Yaskawa INFORM job: A_ROOF_SIDE_0617_2_PAINT_16.JBI

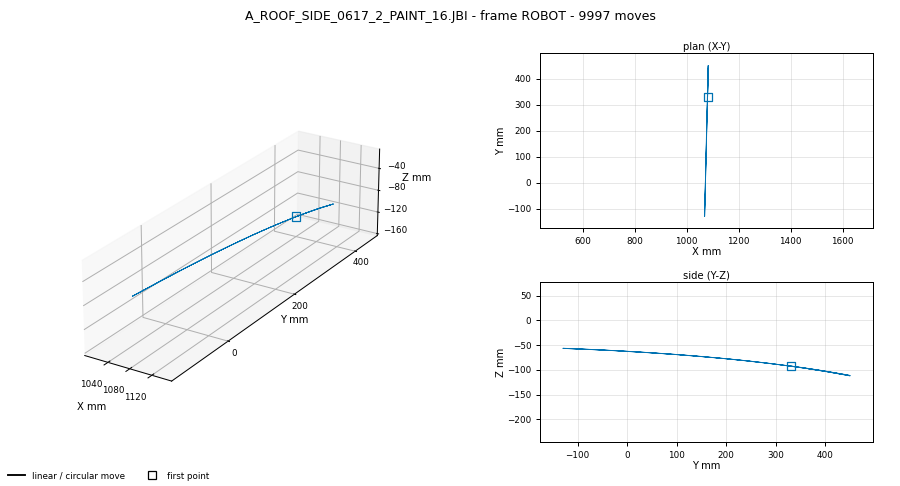
[picture p0: tool path of A_ROOF_SIDE_0617_2_PAINT_16.JBI in frame ROBOT, 9997 of 9997 moves have a stored position in this frame; points joined in program order, loops and branches not executed]
/JOB
//NAME A_ROOF_SIDE_0617_2_PAINT16
//POS
///NPOS 9997,0,0,0,0,0
///TOOL 1
///USER 0
///POSTYPE ROBOT
///RECTAN
///RCONF 1,0,0,0,0,0,0,0,0,0,0,0,0,0,0,0,0,0,0,0,0,0,0,0
C00000=1080.801,330.181,-92.181,175.912,27.090,154.615
C00001=1080.812,330.595,-92.237,175.918,27.097,154.616
C00002=1080.821,331.010,-92.293,175.923,27.105,154.617
C00003=1080.832,331.424,-92.349,175.928,27.113,154.618
C00004=1080.838,331.672,-92.382,175.931,27.117,154.619
C00005=1080.844,331.919,-92.416,175.934,27.122,154.620
C00006=1080.849,332.167,-92.449,175.937,27.126,154.620
C00007=1080.856,332.416,-92.482,175.940,27.131,154.621
C00008=1080.862,332.663,-92.516,175.943,27.136,154.622
C00009=1080.868,332.911,-92.550,175.947,27.141,154.623
C00010=1080.873,333.158,-92.584,175.950,27.146,154.623
C00011=1080.879,333.406,-92.617,175.953,27.150,154.624
C00012=1080.885,333.653,-92.651,175.956,27.155,154.625
C00013=1080.892,333.902,-92.684,175.959,27.160,154.626
C00014=1080.898,334.149,-92.718,175.962,27.165,154.627
C00015=1080.904,334.396,-92.752,175.965,27.170,154.627
C00016=1080.909,334.644,-92.786,175.968,27.174,154.628
C00017=1080.915,334.891,-92.820,175.971,27.179,154.629
C00018=1080.921,335.140,-92.853,175.975,27.183,154.630
C00019=1080.927,335.387,-92.888,175.978,27.188,154.630
C00020=1080.933,335.635,-92.922,175.981,27.193,154.631
C00021=1080.939,335.883,-92.955,175.984,27.198,154.632
C00022=1080.946,336.130,-92.989,175.987,27.202,154.633
C00023=1080.951,336.377,-93.023,175.990,27.207,154.633
C00024=1080.957,336.625,-93.056,175.994,27.212,154.634
C00025=1080.963,336.873,-93.091,175.997,27.217,154.635
C00026=1080.969,337.121,-93.125,176.000,27.222,154.636
C00027=1080.975,337.368,-93.159,176.003,27.227,154.637
C00028=1080.981,337.616,-93.192,176.006,27.232,154.637
C00029=1080.987,337.864,-93.226,176.009,27.236,154.638
C00030=1080.993,338.111,-93.260,176.012,27.241,154.639
C00031=1080.999,338.359,-93.295,176.015,27.246,154.640
C00032=1081.005,338.606,-93.329,176.018,27.251,154.641
C00033=1081.011,338.854,-93.363,176.022,27.256,154.642
C00034=1081.018,339.102,-93.397,176.025,27.261,154.642
C00035=1081.024,339.349,-93.431,176.028,27.266,154.643
C00036=1081.029,339.596,-93.466,176.031,27.270,154.644
C00037=1081.035,339.845,-93.500,176.034,27.276,154.645
C00038=1081.041,340.092,-93.534,176.037,27.280,154.646
C00039=1081.047,340.340,-93.568,176.040,27.285,154.646
C00040=1081.053,340.588,-93.602,176.043,27.290,154.647
C00041=1081.059,340.835,-93.636,176.047,27.295,154.648
C00042=1081.065,341.082,-93.671,176.050,27.300,154.649
C00043=1081.071,341.330,-93.706,176.053,27.305,154.650
C00044=1081.077,341.577,-93.740,176.056,27.310,154.650
C00045=1081.083,341.825,-93.775,176.059,27.315,154.651
C00046=1081.089,342.072,-93.809,176.062,27.320,154.652
C00047=1081.095,342.320,-93.843,176.065,27.325,154.653
C00048=1081.101,342.568,-93.877,176.069,27.330,154.654
C00049=1081.106,342.815,-93.912,176.072,27.335,154.655
C00050=1081.113,343.063,-93.946,176.075,27.340,154.655
C00051=1081.119,343.310,-93.981,176.078,27.345,154.656
C00052=1081.129,343.719,-94.038,176.084,27.353,154.658
C00053=1081.140,344.129,-94.095,176.089,27.362,154.659
C00054=1081.149,344.538,-94.152,176.095,27.370,154.660
C00055=1081.159,344.947,-94.210,176.100,27.379,154.662
C00056=1081.165,345.194,-94.244,176.103,27.383,154.663
C00057=1081.171,345.442,-94.280,176.106,27.389,154.664
C00058=1081.177,345.689,-94.314,176.109,27.394,154.665
C00059=1081.183,345.937,-94.349,176.113,27.399,154.665
C00060=1081.189,346.184,-94.383,176.116,27.404,154.666
C00061=1081.195,346.432,-94.418,176.119,27.409,154.667
C00062=1081.201,346.679,-94.453,176.122,27.414,154.668
C00063=1081.207,346.927,-94.488,176.125,27.419,154.669
C00064=1081.213,347.174,-94.523,176.129,27.425,154.670
C00065=1081.219,347.422,-94.557,176.132,27.430,154.671
C00066=1081.225,347.669,-94.593,176.135,27.435,154.671
C00067=1081.231,347.917,-94.627,176.138,27.440,154.672
C00068=1081.237,348.164,-94.663,176.142,27.446,154.673
C00069=1081.243,348.412,-94.697,176.145,27.451,154.674
C00070=1081.250,348.659,-94.732,176.148,27.456,154.675
C00071=1081.255,348.906,-94.767,176.151,27.461,154.676
C00072=1081.261,349.154,-94.802,176.154,27.466,154.677
C00073=1081.267,349.401,-94.837,176.158,27.472,154.678
C00074=1081.273,349.649,-94.873,176.161,27.477,154.679
C00075=1081.280,349.897,-94.907,176.164,27.482,154.680
C00076=1081.285,350.144,-94.943,176.167,27.488,154.680
C00077=1081.292,350.391,-94.978,176.171,27.493,154.681
C00078=1081.298,350.639,-95.013,176.174,27.498,154.682
C00079=1081.304,350.886,-95.048,176.177,27.504,154.683
C00080=1081.310,351.134,-95.083,176.181,27.509,154.684
C00081=1081.317,351.381,-95.118,176.184,27.514,154.685
C00082=1081.322,351.628,-95.154,176.187,27.519,154.686
C00083=1081.328,351.876,-95.189,176.190,27.525,154.687
C00084=1081.334,352.124,-95.224,176.194,27.530,154.688
C00085=1081.340,352.371,-95.259,176.197,27.535,154.689
C00086=1081.347,352.618,-95.294,176.200,27.541,154.689
C00087=1081.353,352.866,-95.330,176.203,27.546,154.690
C00088=1081.359,353.113,-95.366,176.207,27.552,154.691
C00089=1081.364,353.360,-95.401,176.210,27.557,154.692
C00090=1081.371,353.608,-95.436,176.213,27.562,154.693
C00091=1081.377,353.855,-95.472,176.217,27.568,154.694
C00092=1081.382,354.102,-95.508,176.220,27.573,154.695
C00093=1081.388,354.350,-95.543,176.223,27.579,154.696
C00094=1081.395,354.597,-95.578,176.227,27.584,154.697
C00095=1081.401,354.845,-95.614,176.229,27.590,154.698
C00096=1081.407,355.092,-95.650,176.232,27.595,154.699
C00097=1081.413,355.340,-95.685,176.236,27.601,154.700
C00098=1081.419,355.587,-95.721,176.239,27.606,154.701
C00099=1081.425,355.835,-95.756,176.242,27.612,154.702
C00100=1081.431,356.081,-95.792,176.246,27.617,154.703
C00101=1081.437,356.329,-95.828,176.249,27.622,154.704
C00102=1081.443,356.576,-95.864,176.252,27.628,154.705
C00103=1081.449,356.824,-95.899,176.256,27.634,154.706
C00104=1081.459,357.236,-95.959,176.261,27.643,154.707
C00105=1081.470,357.647,-96.019,176.267,27.652,154.709
C00106=1081.480,358.060,-96.078,176.272,27.661,154.711
C00107=1081.490,358.472,-96.138,176.278,27.671,154.712
C00108=1081.496,358.720,-96.174,176.281,27.676,154.713
C00109=1081.503,358.967,-96.210,176.284,27.682,154.714
C00110=1081.509,359.214,-96.245,176.288,27.688,154.715
C00111=1081.515,359.461,-96.281,176.291,27.693,154.716
C00112=1081.521,359.708,-96.317,176.294,27.699,154.717
C00113=1081.527,359.955,-96.353,176.298,27.705,154.718
C00114=1081.533,360.203,-96.389,176.301,27.711,154.719
C00115=1081.540,360.450,-96.426,176.305,27.717,154.720
C00116=1081.546,360.698,-96.461,176.308,27.722,154.721
C00117=1081.552,360.945,-96.498,176.311,27.727,154.722
C00118=1081.558,361.193,-96.533,176.315,27.733,154.723
C00119=1081.564,361.440,-96.570,176.318,27.739,154.724
C00120=1081.570,361.688,-96.606,176.322,27.745,154.725
C00121=1081.576,361.935,-96.643,176.324,27.751,154.726
C00122=1081.582,362.181,-96.679,176.327,27.756,154.727
C00123=1081.588,362.429,-96.714,176.331,27.762,154.728
C00124=1081.594,362.676,-96.751,176.334,27.768,154.729
C00125=1081.601,362.923,-96.787,176.338,27.774,154.730
C00126=1081.607,363.170,-96.823,176.341,27.780,154.731
C00127=1081.613,363.417,-96.860,176.344,27.785,154.733
C00128=1081.619,363.665,-96.896,176.348,27.792,154.734
C00129=1081.626,363.912,-96.932,176.351,27.797,154.735
C00130=1081.631,364.160,-96.969,176.355,27.803,154.736
C00131=1081.637,364.407,-97.005,176.358,27.809,154.737
C00132=1081.644,364.654,-97.042,176.362,27.815,154.738
C00133=1081.650,364.901,-97.078,176.365,27.821,154.739
C00134=1081.657,365.148,-97.115,176.369,27.827,154.740
C00135=1081.663,365.396,-97.151,176.372,27.833,154.741
C00136=1081.669,365.643,-97.188,176.374,27.839,154.742
C00137=1081.675,365.891,-97.224,176.378,27.845,154.743
C00138=1081.681,366.138,-97.261,176.381,27.850,154.744
C00139=1081.687,366.385,-97.298,176.385,27.857,154.745
C00140=1081.693,366.632,-97.334,176.388,27.862,154.746
C00141=1081.699,366.879,-97.371,176.392,27.869,154.748
C00142=1081.705,367.126,-97.408,176.395,27.875,154.749
C00143=1081.712,367.373,-97.445,176.399,27.881,154.750
C00144=1081.717,367.620,-97.482,176.402,27.887,154.751
C00145=1081.724,367.867,-97.518,176.406,27.893,154.752
C00146=1081.730,368.114,-97.555,176.409,27.899,154.753
C00147=1081.736,368.362,-97.592,176.412,27.906,154.754
C00148=1081.742,368.609,-97.628,176.415,27.911,154.755
C00149=1081.748,368.857,-97.666,176.419,27.918,154.756
C00150=1081.755,369.103,-97.703,176.422,27.924,154.758
C00151=1081.761,369.350,-97.739,176.426,27.930,154.759
C00152=1081.767,369.598,-97.776,176.429,27.936,154.760
C00153=1081.773,369.845,-97.813,176.433,27.942,154.761
C00154=1081.779,370.092,-97.850,176.436,27.948,154.762
C00155=1081.786,370.339,-97.887,176.440,27.955,154.763
C00156=1081.791,370.553,-97.919,176.443,27.960,154.764
C00157=1081.796,370.767,-97.950,176.446,27.966,154.765
C00158=1081.801,370.981,-97.983,176.448,27.970,154.766
C00159=1081.807,371.195,-98.015,176.451,27.976,154.767
C00160=1081.812,371.409,-98.047,176.454,27.981,154.768
C00161=1081.818,371.623,-98.080,176.457,27.987,154.769
C00162=1081.823,371.837,-98.112,176.460,27.992,154.770
C00163=1081.828,372.052,-98.144,176.463,27.998,154.771
C00164=1081.835,372.299,-98.181,176.467,28.004,154.772
C00165=1081.841,372.546,-98.218,176.470,28.010,154.773
C00166=1081.847,372.792,-98.255,176.474,28.016,154.775
C00167=1081.854,373.041,-98.293,176.477,28.023,154.776
C00168=1081.860,373.287,-98.330,176.480,28.030,154.777
C00169=1081.866,373.534,-98.367,176.483,28.036,154.778
C00170=1081.873,373.781,-98.404,176.487,28.042,154.779
C00171=1081.879,374.028,-98.442,176.491,28.048,154.781
C00172=1081.885,374.276,-98.479,176.494,28.055,154.782
C00173=1081.891,374.522,-98.516,176.498,28.061,154.783
C00174=1081.898,374.769,-98.555,176.501,28.068,154.784
C00175=1081.903,375.017,-98.592,176.505,28.074,154.785
C00176=1081.909,375.264,-98.629,176.508,28.081,154.787
C00177=1081.916,375.510,-98.667,176.511,28.087,154.788
C00178=1081.922,375.757,-98.705,176.515,28.094,154.789
C00179=1081.928,376.005,-98.742,176.518,28.100,154.790
C00180=1081.934,376.252,-98.779,176.522,28.107,154.792
C00181=1081.941,376.499,-98.817,176.526,28.114,154.793
C00182=1081.947,376.745,-98.855,176.529,28.120,154.794
C00183=1081.953,376.992,-98.892,176.533,28.127,154.795
C00184=1081.960,377.240,-98.931,176.535,28.133,154.797
C00185=1081.965,377.487,-98.968,176.539,28.140,154.798
C00186=1081.972,377.733,-99.005,176.543,28.146,154.799
C00187=1081.978,377.981,-99.043,176.546,28.153,154.800
C00188=1081.984,378.228,-99.081,176.550,28.160,154.802
C00189=1081.991,378.475,-99.119,176.554,28.167,154.803
C00190=1081.997,378.722,-99.157,176.557,28.173,154.804
C00191=1082.004,378.969,-99.194,176.560,28.180,154.805
C00192=1082.010,379.216,-99.232,176.564,28.187,154.807
C00193=1082.016,379.462,-99.270,176.567,28.193,154.808
C00194=1082.022,379.709,-99.308,176.571,28.200,154.809
C00195=1082.028,379.956,-99.346,176.575,28.207,154.810
C00196=1082.035,380.203,-99.384,176.578,28.214,154.812
C00197=1082.041,380.450,-99.422,176.582,28.220,154.813
C00198=1082.048,380.697,-99.460,176.585,28.227,154.814
C00199=1082.054,380.944,-99.497,176.588,28.234,154.816
C00200=1082.061,381.191,-99.536,176.592,28.241,154.817
C00201=1082.067,381.438,-99.574,176.596,28.248,154.818
C00202=1082.073,381.685,-99.612,176.599,28.255,154.820
C00203=1082.080,381.932,-99.650,176.603,28.261,154.821
C00204=1082.086,382.179,-99.689,176.606,28.268,154.822
C00205=1082.092,382.426,-99.727,176.610,28.275,154.823
C00206=1082.098,382.673,-99.765,176.613,28.282,154.825
C00207=1082.105,382.920,-99.803,176.617,28.289,154.826
C00208=1082.111,383.166,-99.841,176.621,28.296,154.827
C00209=1082.118,383.413,-99.880,176.624,28.303,154.829
C00210=1082.123,383.660,-99.918,176.627,28.310,154.830
C00211=1082.130,383.907,-99.957,176.631,28.318,154.832
C00212=1082.136,384.135,-99.993,176.634,28.324,154.833
C00213=1082.141,384.364,-100.028,176.638,28.330,154.834
C00214=1082.148,384.592,-100.063,176.641,28.337,154.835
C00215=1082.153,384.819,-100.099,176.644,28.344,154.837
C00216=1082.159,385.048,-100.135,176.648,28.350,154.838
C00217=1082.165,385.276,-100.170,176.651,28.356,154.839
C00218=1082.171,385.505,-100.206,176.655,28.363,154.840
C00219=1082.177,385.733,-100.241,176.658,28.370,154.842
C00220=1082.182,385.980,-100.280,176.661,28.377,154.843
C00221=1082.189,386.227,-100.319,176.665,28.385,154.844
C00222=1082.195,386.474,-100.357,176.668,28.392,154.846
C00223=1082.201,386.721,-100.395,176.672,28.399,154.847
C00224=1082.208,386.967,-100.434,176.676,28.406,154.849
C00225=1082.214,387.214,-100.473,176.680,28.413,154.850
C00226=1082.220,387.461,-100.512,176.683,28.421,154.852
C00227=1082.227,387.708,-100.550,176.686,28.428,154.853
C00228=1082.234,387.955,-100.589,176.690,28.435,154.854
C00229=1082.240,388.202,-100.628,176.694,28.442,154.856
C00230=1082.246,388.448,-100.667,176.698,28.450,154.857
C00231=1082.253,388.695,-100.706,176.701,28.458,154.859
C00232=1082.260,388.942,-100.744,176.705,28.465,154.860
C00233=1082.266,389.189,-100.784,176.708,28.472,154.862
C00234=1082.272,389.435,-100.822,176.712,28.479,154.863
C00235=1082.279,389.682,-100.861,176.716,28.487,154.865
C00236=1082.285,389.929,-100.901,176.719,28.494,154.866
C00237=1082.292,390.176,-100.939,176.723,28.502,154.867
C00238=1082.298,390.423,-100.978,176.727,28.509,154.869
C00239=1082.304,390.669,-101.017,176.731,28.517,154.870
C00240=1082.311,390.916,-101.056,176.734,28.524,154.872
C00241=1082.318,391.163,-101.095,176.738,28.531,154.873
C00242=1082.324,391.410,-101.134,176.741,28.539,154.875
C00243=1082.330,391.657,-101.173,176.745,28.546,154.876
C00244=1082.338,391.903,-101.213,176.749,28.554,154.878
C00245=1082.344,392.150,-101.252,176.753,28.562,154.879
C00246=1082.350,392.396,-101.291,176.756,28.570,154.881
C00247=1082.356,392.643,-101.330,176.760,28.578,154.882
C00248=1082.362,392.890,-101.370,176.763,28.585,154.884
C00249=1082.369,393.137,-101.409,176.767,28.593,154.885
C00250=1082.375,393.384,-101.449,176.771,28.601,154.887
C00251=1082.382,393.630,-101.488,176.774,28.608,154.888
C00252=1082.388,393.877,-101.528,176.778,28.616,154.890
C00253=1082.395,394.124,-101.566,176.782,28.624,154.892
C00254=1082.402,394.370,-101.607,176.786,28.632,154.893
C00255=1082.408,394.618,-101.646,176.790,28.639,154.895
C00256=1082.415,394.864,-101.686,176.793,28.647,154.896
C00257=1082.421,395.111,-101.725,176.797,28.655,154.898
C00258=1082.427,395.357,-101.765,176.801,28.663,154.899
C00259=1082.434,395.604,-101.804,176.805,28.671,154.901
C00260=1082.440,395.851,-101.844,176.808,28.679,154.903
C00261=1082.446,396.098,-101.884,176.812,28.687,154.904
C00262=1082.453,396.344,-101.924,176.816,28.695,154.906
C00263=1082.460,396.591,-101.963,176.819,28.703,154.907
C00264=1082.466,396.838,-102.003,176.823,28.711,154.909
C00265=1082.472,397.084,-102.043,176.826,28.719,154.911
C00266=1082.479,397.331,-102.082,176.830,28.727,154.912
C00267=1082.486,397.578,-102.122,176.834,28.735,154.914
C00268=1082.491,397.813,-102.161,176.838,28.743,154.915
C00269=1082.498,398.048,-102.198,176.842,28.750,154.917
C00270=1082.504,398.283,-102.236,176.845,28.759,154.919
C00271=1082.510,398.519,-102.275,176.848,28.766,154.920
C00272=1082.517,398.754,-102.313,176.852,28.774,154.922
C00273=1082.523,398.989,-102.350,176.856,28.782,154.923
C00274=1082.529,399.224,-102.389,176.860,28.790,154.925
C00275=1082.536,399.461,-102.427,176.863,28.798,154.926
C00276=1082.542,399.707,-102.467,176.867,28.806,154.928
C00277=1082.548,399.954,-102.507,176.871,28.814,154.930
C00278=1082.555,400.200,-102.547,176.875,28.823,154.932
C00279=1082.561,400.447,-102.587,176.878,28.831,154.933
C00280=1082.568,400.693,-102.628,176.882,28.840,154.935
C00281=1082.575,400.940,-102.668,176.886,28.848,154.937
C00282=1082.581,401.187,-102.708,176.890,28.856,154.938
C00283=1082.587,401.433,-102.748,176.893,28.865,154.940
C00284=1082.594,401.680,-102.789,176.897,28.873,154.942
C00285=1082.601,401.927,-102.829,176.901,28.882,154.944
C00286=1082.607,402.174,-102.869,176.905,28.890,154.945
C00287=1082.614,402.420,-102.910,176.908,28.898,154.947
C00288=1082.621,402.667,-102.951,176.913,28.907,154.949
C00289=1082.627,402.913,-102.991,176.917,28.916,154.950
C00290=1082.633,403.160,-103.031,176.921,28.924,154.952
C00291=1082.641,403.406,-103.072,176.924,28.933,154.954
C00292=1082.646,403.653,-103.113,176.928,28.942,154.956
C00293=1082.653,403.900,-103.153,176.932,28.950,154.958
C00294=1082.660,404.147,-103.193,176.936,28.959,154.959
C00295=1082.666,404.393,-103.234,176.939,28.968,154.961
C00296=1082.673,404.639,-103.274,176.944,28.976,154.963
C00297=1082.680,404.886,-103.316,176.948,28.985,154.965
C00298=1082.686,405.133,-103.356,176.952,28.994,154.967
C00299=1082.692,405.379,-103.397,176.955,29.002,154.968
C00300=1082.699,405.626,-103.438,176.959,29.012,154.970
C00301=1082.706,405.872,-103.478,176.964,29.021,154.972
C00302=1082.712,406.119,-103.520,176.968,29.030,154.974
C00303=1082.719,406.365,-103.561,176.971,29.038,154.976
C00304=1082.726,406.612,-103.601,176.975,29.047,154.978
C00305=1082.733,406.858,-103.642,176.979,29.056,154.980
C00306=1082.738,407.105,-103.683,176.983,29.065,154.981
C00307=1082.746,407.352,-103.724,176.987,29.074,154.983
C00308=1082.752,407.598,-103.765,176.991,29.083,154.985
C00309=1082.759,407.845,-103.807,176.995,29.092,154.987
C00310=1082.765,408.091,-103.847,176.999,29.102,154.989
C00311=1082.772,408.338,-103.889,177.003,29.111,154.991
C00312=1082.778,408.584,-103.930,177.007,29.120,154.993
C00313=1082.785,408.831,-103.971,177.011,29.129,154.995
C00314=1082.791,409.077,-104.012,177.015,29.139,154.997
C00315=1082.798,409.324,-104.053,177.019,29.148,154.999
C00316=1082.805,409.570,-104.094,177.023,29.157,155.001
C00317=1082.811,409.817,-104.136,177.027,29.167,155.003
C00318=1082.818,410.064,-104.177,177.031,29.176,155.004
C00319=1082.824,410.310,-104.219,177.035,29.185,155.006
C00320=1082.832,410.556,-104.260,177.040,29.195,155.008
C00321=1082.838,410.803,-104.301,177.043,29.204,155.010
C00322=1082.845,411.049,-104.343,177.047,29.213,155.012
C00323=1082.851,411.296,-104.384,177.052,29.223,155.014
C00324=1082.858,411.532,-104.424,177.056,29.232,155.016
C00325=1082.864,411.768,-104.464,177.059,29.241,155.018
C00326=1082.871,412.005,-104.504,177.063,29.250,155.020
C00327=1082.877,412.241,-104.544,177.067,29.260,155.022
C00328=1082.884,412.477,-104.583,177.072,29.269,155.024
C00329=1082.891,412.713,-104.624,177.075,29.278,155.026
C00330=1082.897,412.949,-104.663,177.079,29.287,155.028
C00331=1082.903,413.186,-104.703,177.083,29.296,155.030
C00332=1082.910,413.432,-104.746,177.088,29.306,155.032
C00333=1082.917,413.678,-104.787,177.091,29.316,155.034
C00334=1082.923,413.925,-104.828,177.096,29.326,155.036
C00335=1082.931,414.171,-104.870,177.100,29.335,155.038
C00336=1082.937,414.418,-104.912,177.104,29.345,155.040
C00337=1082.944,414.664,-104.955,177.108,29.355,155.042
C00338=1082.951,414.910,-104.995,177.112,29.365,155.044
C00339=1082.958,415.156,-105.038,177.117,29.375,155.046
C00340=1082.964,415.403,-105.080,177.120,29.384,155.048
C00341=1082.972,415.649,-105.122,177.125,29.394,155.051
C00342=1082.979,415.896,-105.164,177.129,29.404,155.053
C00343=1082.985,416.142,-105.206,177.134,29.414,155.055
C00344=1082.992,416.389,-105.248,177.137,29.424,155.057
C00345=1082.998,416.635,-105.290,177.142,29.435,155.059
C00346=1083.005,416.881,-105.333,177.147,29.445,155.061
C00347=1083.013,417.127,-105.375,177.150,29.455,155.063
C00348=1083.019,417.374,-105.416,177.155,29.465,155.066
C00349=1083.026,417.620,-105.459,177.159,29.476,155.068
C00350=1083.033,417.867,-105.502,177.163,29.486,155.070
C00351=1083.040,418.113,-105.544,177.167,29.496,155.072
C00352=1083.046,418.359,-105.586,177.172,29.506,155.074
C00353=1083.053,418.605,-105.629,177.177,29.517,155.077
C00354=1083.060,418.851,-105.671,177.180,29.527,155.079
C00355=1083.066,419.098,-105.713,177.185,29.538,155.081
C00356=1083.073,419.344,-105.756,177.190,29.548,155.083
C00357=1083.080,419.591,-105.798,177.193,29.558,155.086
C00358=1083.087,419.836,-105.842,177.198,29.569,155.088
C00359=1083.094,420.083,-105.884,177.202,29.580,155.090
C00360=1083.101,420.329,-105.927,177.207,29.590,155.092
C00361=1083.108,420.575,-105.969,177.211,29.600,155.095
C00362=1083.115,420.821,-106.012,177.215,29.611,155.097
C00363=1083.121,421.068,-106.054,177.220,29.622,155.099
C00364=1083.129,421.315,-106.097,177.224,29.632,155.102
C00365=1083.136,421.560,-106.140,177.229,29.644,155.104
C00366=1083.143,421.807,-106.183,177.233,29.654,155.106
C00367=1083.150,422.053,-106.225,177.238,29.665,155.109
C00368=1083.157,422.299,-106.269,177.242,29.676,155.111
C00369=1083.164,422.545,-106.311,177.247,29.687,155.113
C00370=1083.171,422.791,-106.354,177.251,29.698,155.116
C00371=1083.177,423.037,-106.398,177.255,29.708,155.118
C00372=1083.184,423.283,-106.440,177.260,29.719,155.120
C00373=1083.191,423.529,-106.483,177.265,29.731,155.123
C00374=1083.199,423.776,-106.526,177.268,29.741,155.125
C00375=1083.205,424.022,-106.570,177.273,29.753,155.128
C00376=1083.212,424.268,-106.613,177.278,29.764,155.130
C00377=1083.219,424.514,-106.656,177.283,29.775,155.133
C00378=1083.225,424.760,-106.700,177.287,29.786,155.135
C00379=1083.233,425.007,-106.743,177.291,29.797,155.138
C00380=1083.240,425.254,-106.787,177.296,29.809,155.140
C00381=1083.247,425.501,-106.830,177.300,29.820,155.142
C00382=1083.254,425.748,-106.873,177.305,29.831,155.145
C00383=1083.261,425.995,-106.917,177.310,29.843,155.147
C00384=1083.268,426.241,-106.960,177.315,29.854,155.150
C00385=1083.275,426.487,-107.003,177.319,29.866,155.152
C00386=1083.282,426.733,-107.048,177.324,29.877,155.155
C00387=1083.289,426.979,-107.091,177.329,29.888,155.157
C00388=1083.296,427.225,-107.134,177.332,29.900,155.160
C00389=1083.304,427.471,-107.178,177.337,29.911,155.163
C00390=1083.311,427.717,-107.222,177.342,29.923,155.165
C00391=1083.317,427.963,-107.265,177.347,29.935,155.168
C00392=1083.325,428.209,-107.309,177.351,29.947,155.170
C00393=1083.332,428.455,-107.352,177.356,29.958,155.173
C00394=1083.339,428.702,-107.397,177.361,29.970,155.175
C00395=1083.345,428.948,-107.440,177.366,29.982,155.178
C00396=1083.353,429.193,-107.484,177.370,29.994,155.181
C00397=1083.360,429.439,-107.529,177.375,30.006,155.183
C00398=1083.367,429.685,-107.572,177.380,30.018,155.186
C00399=1083.374,429.932,-107.616,177.384,30.030,155.189
C00400=1083.382,430.177,-107.660,177.389,30.042,155.191
C00401=1083.388,430.423,-107.704,177.394,30.054,155.194
C00402=1083.395,430.669,-107.749,177.399,30.066,155.197
C00403=1083.403,430.914,-107.792,177.403,30.078,155.199
C00404=1083.410,431.160,-107.837,177.408,30.090,155.202
C00405=1083.417,431.406,-107.880,177.413,30.102,155.205
C00406=1083.424,431.652,-107.925,177.418,30.114,155.208
C00407=1083.431,431.899,-107.969,177.423,30.127,155.210
C00408=1083.439,432.144,-108.013,177.428,30.139,155.213
C00409=1083.446,432.391,-108.058,177.433,30.152,155.216
C00410=1083.453,432.636,-108.102,177.438,30.164,155.218
C00411=1083.460,432.882,-108.147,177.442,30.176,155.221
C00412=1083.466,433.128,-108.191,177.447,30.189,155.224
C00413=1083.474,433.374,-108.235,177.452,30.202,155.227
C00414=1083.482,433.620,-108.280,177.457,30.214,155.230
C00415=1083.489,433.865,-108.325,177.462,30.227,155.233
C00416=1083.496,434.111,-108.370,177.467,30.239,155.235
C00417=1083.503,434.356,-108.414,177.472,30.252,155.238
C00418=1083.510,434.602,-108.459,177.477,30.265,155.241
C00419=1083.517,434.849,-108.504,177.481,30.278,155.244
C00420=1083.524,435.092,-108.548,177.486,30.291,155.247
C00421=1083.531,435.335,-108.592,177.492,30.303,155.250
C00422=1083.538,435.579,-108.637,177.497,30.316,155.253
C00423=1083.545,435.823,-108.681,177.501,30.329,155.256
C00424=1083.553,436.066,-108.726,177.506,30.342,155.259
C00425=1083.560,436.309,-108.770,177.511,30.355,155.261
C00426=1083.567,436.553,-108.815,177.517,30.368,155.264
C00427=1083.575,436.796,-108.860,177.522,30.381,155.267
C00428=1083.582,437.042,-108.905,177.526,30.394,155.270
C00429=1083.589,437.288,-108.950,177.531,30.407,155.273
C00430=1083.596,437.533,-108.995,177.537,30.421,155.276
C00431=1083.604,437.779,-109.040,177.542,30.434,155.279
C00432=1083.611,438.025,-109.085,177.547,30.447,155.283
C00433=1083.619,438.270,-109.130,177.552,30.460,155.285
C00434=1083.626,438.517,-109.175,177.557,30.474,155.289
C00435=1083.634,438.762,-109.221,177.563,30.487,155.292
C00436=1083.644,439.107,-109.284,177.569,30.507,155.296
C00437=1083.655,439.451,-109.348,177.577,30.525,155.300
C00438=1083.665,439.796,-109.412,177.584,30.545,155.305
C00439=1083.676,440.141,-109.476,177.591,30.564,155.309
C00440=1083.683,440.386,-109.521,177.597,30.578,155.312
C00441=1083.690,440.631,-109.567,177.602,30.592,155.315
C00442=1083.697,440.877,-109.612,177.608,30.606,155.319
C00443=1083.704,441.123,-109.658,177.613,30.620,155.322
C00444=1083.712,441.368,-109.704,177.618,30.634,155.325
C00445=1083.720,441.614,-109.750,177.623,30.648,155.328
C00446=1083.727,441.860,-109.796,177.629,30.662,155.332
C00447=1083.735,442.106,-109.841,177.634,30.676,155.335
C00448=1083.743,442.351,-109.887,177.640,30.691,155.338
C00449=1083.749,442.597,-109.933,177.645,30.705,155.342
C00450=1083.757,442.842,-109.980,177.650,30.719,155.345
C00451=1083.764,443.087,-110.026,177.655,30.733,155.348
C00452=1083.772,443.333,-110.072,177.661,30.748,155.351
C00453=1083.780,443.578,-110.117,177.667,30.763,155.355
C00454=1083.786,443.824,-110.163,177.672,30.777,155.358
C00455=1083.795,444.069,-110.210,177.678,30.792,155.362
C00456=1083.802,444.315,-110.256,177.683,30.806,155.365
C00457=1083.810,444.560,-110.303,177.689,30.821,155.368
C00458=1083.817,444.805,-110.348,177.694,30.836,155.372
C00459=1083.825,445.052,-110.395,177.699,30.851,155.375
C00460=1083.833,445.297,-110.441,177.705,30.866,155.379
C00461=1083.840,445.542,-110.488,177.711,30.881,155.382
C00462=1083.847,445.788,-110.535,177.716,30.895,155.386
C00463=1083.856,446.033,-110.581,177.721,30.910,155.389
C00464=1083.862,446.279,-110.628,177.725,30.925,155.393
C00465=1083.870,446.524,-110.674,177.730,30.940,155.396
C00466=1083.878,446.769,-110.721,177.734,30.955,155.400
C00467=1083.885,447.015,-110.768,177.738,30.969,155.403
C00468=1083.893,447.260,-110.814,177.742,30.984,155.407
C00469=1083.901,447.506,-110.861,177.746,30.999,155.410
C00470=1083.909,447.751,-110.908,177.749,31.014,155.414
C00471=1083.917,447.996,-110.955,177.752,31.028,155.418
C00472=1083.924,448.242,-111.002,177.755,31.044,155.421
C00473=1083.932,448.486,-111.048,177.758,31.058,155.425
C00474=1083.940,448.732,-111.096,177.760,31.073,155.428
C00475=1083.947,448.977,-111.143,177.763,31.088,155.432
C00476=1083.955,449.222,-111.189,177.765,31.102,155.436
C00477=1083.963,449.468,-111.236,177.767,31.117,155.439
C00478=1083.973,449.712,-111.281,177.770,31.130,155.443
C00479=1083.985,449.959,-111.326,177.772,31.143,155.446
C00480=1083.614,449.951,-111.536,177.739,31.321,155.494
C00481=1083.601,449.705,-111.492,177.737,31.309,155.490
C00482=1083.591,449.459,-111.446,177.735,31.295,155.487
C00483=1083.583,449.215,-111.400,177.733,31.281,155.483
C00484=1083.575,448.969,-111.353,177.730,31.266,155.480
C00485=1083.567,448.725,-111.306,177.728,31.251,155.476
C00486=1083.559,448.479,-111.258,177.725,31.236,155.473
C00487=1083.552,448.234,-111.211,177.722,31.222,155.469
C00488=1083.544,447.989,-111.165,177.719,31.207,155.465
C00489=1083.536,447.744,-111.118,177.716,31.192,155.462
C00490=1083.529,447.497,-111.071,177.712,31.177,155.458
C00491=1083.521,447.252,-111.025,177.708,31.162,155.454
C00492=1083.513,447.007,-110.977,177.704,31.147,155.451
C00493=1083.506,446.761,-110.930,177.700,31.132,155.447
C00494=1083.497,446.516,-110.884,177.696,31.118,155.444
C00495=1083.490,446.271,-110.837,177.691,31.103,155.440
C00496=1083.483,446.025,-110.791,177.687,31.088,155.437
C00497=1083.475,445.780,-110.744,177.682,31.073,155.433
C00498=1083.468,445.534,-110.697,177.676,31.058,155.430
C00499=1083.460,445.289,-110.651,177.671,31.044,155.426
C00500=1083.453,445.044,-110.604,177.665,31.028,155.423
C00501=1083.444,444.798,-110.557,177.660,31.014,155.419
C00502=1083.437,444.553,-110.511,177.654,30.999,155.416
C00503=1083.429,444.308,-110.465,177.648,30.984,155.412
C00504=1083.421,444.062,-110.419,177.643,30.969,155.409
C00505=1083.414,443.816,-110.373,177.637,30.955,155.406
C00506=1083.406,443.571,-110.326,177.631,30.940,155.402
C00507=1083.399,443.325,-110.280,177.626,30.926,155.399
C00508=1083.392,443.080,-110.234,177.620,30.911,155.396
C00509=1083.384,442.834,-110.187,177.615,30.897,155.392
C00510=1083.376,442.589,-110.141,177.609,30.883,155.389
C00511=1083.369,442.343,-110.096,177.604,30.868,155.386
C00512=1083.362,442.098,-110.049,177.598,30.854,155.382
C00513=1083.354,441.852,-110.004,177.593,30.840,155.379
C00514=1083.346,441.607,-109.958,177.587,30.826,155.376
C00515=1083.340,441.361,-109.912,177.582,30.811,155.372
C00516=1083.332,441.116,-109.866,177.577,30.797,155.369
C00517=1083.324,440.870,-109.821,177.572,30.784,155.366
C00518=1083.317,440.625,-109.775,177.566,30.770,155.363
C00519=1083.310,440.379,-109.729,177.561,30.756,155.360
C00520=1083.302,440.133,-109.683,177.555,30.742,155.357
C00521=1083.292,439.804,-109.622,177.548,30.723,155.352
C00522=1083.282,439.474,-109.561,177.541,30.705,155.348
C00523=1083.272,439.145,-109.500,177.534,30.687,155.344
C00524=1083.262,438.816,-109.440,177.527,30.668,155.340
C00525=1083.254,438.571,-109.394,177.522,30.655,155.337
C00526=1083.247,438.325,-109.348,177.516,30.641,155.334
C00527=1083.239,438.079,-109.303,177.511,30.628,155.331
C00528=1083.232,437.834,-109.258,177.506,30.615,155.327
C00529=1083.224,437.588,-109.213,177.500,30.601,155.324
C00530=1083.217,437.342,-109.168,177.495,30.588,155.321
C00531=1083.209,437.096,-109.122,177.491,30.575,155.318
C00532=1083.202,436.850,-109.077,177.485,30.561,155.315
C00533=1083.195,436.606,-109.032,177.480,30.548,155.312
C00534=1083.188,436.359,-108.987,177.475,30.535,155.309
C00535=1083.180,436.113,-108.942,177.470,30.522,155.306
C00536=1083.173,435.867,-108.897,177.464,30.509,155.303
C00537=1083.165,435.622,-108.852,177.459,30.496,155.301
C00538=1083.159,435.377,-108.807,177.454,30.483,155.298
C00539=1083.151,435.131,-108.762,177.450,30.470,155.295
C00540=1083.144,434.884,-108.717,177.444,30.457,155.292
C00541=1083.137,434.639,-108.673,177.439,30.445,155.289
C00542=1083.130,434.393,-108.628,177.434,30.432,155.286
C00543=1083.123,434.147,-108.583,177.429,30.419,155.283
C00544=1083.116,433.902,-108.538,177.424,30.406,155.280
C00545=1083.108,433.656,-108.494,177.420,30.394,155.277
C00546=1083.100,433.410,-108.449,177.414,30.381,155.275
C00547=1083.094,433.164,-108.404,177.409,30.368,155.272
C00548=1083.087,432.918,-108.360,177.404,30.356,155.269
C00549=1083.080,432.672,-108.315,177.399,30.343,155.266
C00550=1083.073,432.426,-108.271,177.394,30.331,155.263
C00551=1083.065,432.181,-108.226,177.390,30.318,155.261
C00552=1083.058,431.935,-108.182,177.385,30.306,155.258
C00553=1083.051,431.689,-108.137,177.380,30.294,155.255
C00554=1083.043,431.443,-108.093,177.375,30.282,155.252
C00555=1083.036,431.197,-108.049,177.370,30.269,155.250
C00556=1083.029,430.951,-108.004,177.365,30.257,155.247
C00557=1083.022,430.705,-107.961,177.360,30.245,155.244
C00558=1083.014,430.459,-107.916,177.355,30.233,155.242
C00559=1083.008,430.213,-107.872,177.350,30.221,155.239
C00560=1083.000,429.967,-107.828,177.345,30.209,155.236
C00561=1082.994,429.721,-107.784,177.340,30.197,155.233
C00562=1082.986,429.475,-107.740,177.336,30.185,155.231
C00563=1082.979,429.230,-107.696,177.331,30.173,155.228
C00564=1082.972,428.984,-107.653,177.326,30.161,155.225
C00565=1082.965,428.737,-107.608,177.321,30.149,155.223
C00566=1082.958,428.491,-107.565,177.317,30.137,155.220
C00567=1082.951,428.245,-107.521,177.313,30.126,155.218
C00568=1082.944,428.000,-107.476,177.308,30.114,155.215
C00569=1082.936,427.753,-107.433,177.303,30.102,155.212
C00570=1082.929,427.508,-107.390,177.298,30.090,155.210
C00571=1082.923,427.262,-107.346,177.293,30.079,155.207
C00572=1082.915,427.015,-107.302,177.289,30.067,155.205
C00573=1082.908,426.770,-107.259,177.284,30.056,155.202
C00574=1082.901,426.525,-107.215,177.279,30.044,155.200
C00575=1082.894,426.280,-107.172,177.274,30.033,155.197
C00576=1082.887,426.035,-107.128,177.270,30.022,155.195
C00577=1082.880,425.790,-107.085,177.266,30.010,155.192
C00578=1082.873,425.546,-107.042,177.261,29.999,155.190
C00579=1082.865,425.301,-106.999,177.256,29.988,155.187
C00580=1082.859,425.056,-106.956,177.251,29.977,155.185
C00581=1082.852,424.810,-106.912,177.246,29.965,155.182
C00582=1082.845,424.563,-106.869,177.243,29.954,155.180
C00583=1082.838,424.317,-106.826,177.238,29.943,155.177
C00584=1082.831,424.072,-106.783,177.233,29.932,155.175
C00585=1082.824,423.826,-106.739,177.228,29.921,155.173
C00586=1082.817,423.579,-106.697,177.223,29.909,155.170
C00587=1082.810,423.333,-106.653,177.220,29.899,155.168
C00588=1082.803,423.087,-106.610,177.215,29.887,155.165
C00589=1082.796,422.841,-106.567,177.210,29.876,155.163
C00590=1082.789,422.594,-106.524,177.205,29.866,155.161
C00591=1082.782,422.349,-106.481,177.202,29.855,155.158
C00592=1082.775,422.102,-106.438,177.197,29.843,155.156
C00593=1082.764,421.711,-106.369,177.190,29.827,155.152
C00594=1082.753,421.319,-106.302,177.183,29.809,155.148
C00595=1082.742,420.927,-106.234,177.176,29.793,155.145
C00596=1082.731,420.536,-106.165,177.169,29.775,155.141
C00597=1082.724,420.289,-106.123,177.164,29.765,155.139
C00598=1082.717,420.043,-106.080,177.159,29.754,155.136
C00599=1082.710,419.797,-106.038,177.155,29.744,155.134
C00600=1082.703,419.551,-105.995,177.150,29.733,155.132
C00601=1082.696,419.304,-105.953,177.147,29.723,155.130
C00602=1082.690,419.058,-105.910,177.142,29.712,155.127
C00603=1082.683,418.812,-105.868,177.137,29.702,155.125
C00604=1082.676,418.565,-105.825,177.133,29.691,155.123
C00605=1082.669,418.319,-105.782,177.129,29.681,155.121
C00606=1082.662,418.073,-105.740,177.124,29.670,155.118
C00607=1082.655,417.827,-105.697,177.120,29.660,155.116
C00608=1082.648,417.580,-105.655,177.115,29.650,155.114
C00609=1082.642,417.334,-105.612,177.111,29.640,155.112
C00610=1082.635,417.088,-105.570,177.107,29.629,155.110
C00611=1082.628,416.842,-105.529,177.103,29.619,155.108
C00612=1082.621,416.596,-105.486,177.098,29.609,155.105
C00613=1082.614,416.349,-105.444,177.094,29.599,155.103
C00614=1082.607,416.103,-105.401,177.090,29.589,155.101
C00615=1082.601,415.856,-105.359,177.086,29.579,155.099
C00616=1082.594,415.610,-105.317,177.081,29.569,155.097
C00617=1082.586,415.364,-105.275,177.077,29.559,155.095
C00618=1082.581,415.118,-105.233,177.072,29.549,155.093
C00619=1082.574,414.871,-105.191,177.069,29.539,155.090
C00620=1082.566,414.625,-105.150,177.064,29.530,155.088
C00621=1082.560,414.378,-105.107,177.060,29.519,155.086
C00622=1082.553,414.132,-105.065,177.055,29.510,155.084
C00623=1082.545,413.886,-105.023,177.052,29.500,155.082
C00624=1082.539,413.639,-104.982,177.047,29.490,155.080
C00625=1082.532,413.393,-104.941,177.043,29.481,155.078
C00626=1082.525,413.147,-104.898,177.039,29.471,155.076
C00627=1082.519,412.900,-104.856,177.034,29.461,155.074
C00628=1082.512,412.654,-104.815,177.031,29.452,155.072
C00629=1082.503,412.325,-104.759,177.025,29.439,155.069
C00630=1082.494,411.997,-104.704,177.019,29.426,155.067
C00631=1082.484,411.669,-104.648,177.014,29.413,155.064
C00632=1082.476,411.340,-104.593,177.008,29.401,155.061
C00633=1082.469,411.093,-104.551,177.004,29.391,155.059
C00634=1082.462,410.848,-104.511,177.000,29.382,155.057
C00635=1082.456,410.601,-104.469,176.996,29.372,155.055
C00636=1082.449,410.355,-104.428,176.992,29.363,155.053
C00637=1082.442,410.108,-104.385,176.987,29.353,155.051
C00638=1082.435,409.862,-104.344,176.983,29.344,155.049
C00639=1082.429,409.616,-104.303,176.980,29.335,155.047
C00640=1082.422,409.368,-104.262,176.975,29.325,155.045
C00641=1082.416,409.122,-104.221,176.971,29.316,155.043
C00642=1082.409,408.876,-104.180,176.967,29.307,155.041
C00643=1082.403,408.629,-104.138,176.964,29.298,155.040
C00644=1082.396,408.383,-104.097,176.959,29.288,155.038
C00645=1082.389,408.137,-104.056,176.955,29.279,155.036
C00646=1082.382,407.890,-104.014,176.951,29.270,155.034
C00647=1082.376,407.644,-103.974,176.947,29.261,155.032
C00648=1082.370,407.397,-103.932,176.943,29.252,155.030
C00649=1082.363,407.151,-103.891,176.939,29.243,155.028
C00650=1082.356,406.904,-103.850,176.935,29.234,155.026
C00651=1082.350,406.657,-103.809,176.931,29.225,155.024
C00652=1082.343,406.411,-103.768,176.928,29.216,155.022
C00653=1082.336,406.164,-103.728,176.923,29.206,155.020
C00654=1082.330,405.917,-103.686,176.919,29.198,155.019
C00655=1082.323,405.671,-103.645,176.915,29.189,155.017
C00656=1082.316,405.424,-103.605,176.911,29.180,155.015
C00657=1082.309,405.178,-103.564,176.908,29.171,155.013
C00658=1082.303,404.931,-103.523,176.903,29.162,155.011
C00659=1082.296,404.685,-103.482,176.899,29.153,155.010
C00660=1082.290,404.438,-103.442,176.895,29.145,155.008
C00661=1082.283,404.191,-103.401,176.891,29.136,155.006
C00662=1082.276,403.945,-103.360,176.888,29.127,155.004
C00663=1082.270,403.698,-103.319,176.884,29.119,155.002
C00664=1082.264,403.451,-103.279,176.880,29.110,155.001
C00665=1082.257,403.205,-103.238,176.875,29.101,154.999
C00666=1082.250,402.958,-103.198,176.871,29.092,154.997
C00667=1082.244,402.712,-103.158,176.868,29.084,154.995
C00668=1082.237,402.466,-103.117,176.864,29.076,154.994
C00669=1082.230,402.218,-103.076,176.860,29.067,154.992
C00670=1082.224,401.972,-103.036,176.856,29.058,154.990
C00671=1082.217,401.725,-102.996,176.852,29.050,154.988
C00672=1082.211,401.479,-102.956,176.849,29.041,154.986
C00673=1082.204,401.232,-102.915,176.845,29.033,154.985
C00674=1082.198,400.985,-102.875,176.841,29.025,154.983
C00675=1082.191,400.739,-102.834,176.837,29.016,154.981
C00676=1082.184,400.493,-102.794,176.833,29.008,154.980
C00677=1082.177,400.246,-102.754,176.830,28.999,154.978
C00678=1082.171,399.999,-102.713,176.826,28.991,154.976
C00679=1082.165,399.753,-102.673,176.822,28.983,154.974
C00680=1082.158,399.506,-102.633,176.817,28.974,154.973
C00681=1082.152,399.270,-102.595,176.814,28.966,154.971
C00682=1082.145,399.034,-102.557,176.810,28.958,154.970
C00683=1082.140,398.798,-102.519,176.807,28.951,154.968
C00684=1082.134,398.562,-102.480,176.803,28.943,154.966
C00685=1082.127,398.326,-102.442,176.800,28.935,154.965
C00686=1082.121,398.090,-102.404,176.796,28.927,154.963
C00687=1082.114,397.854,-102.366,176.792,28.919,154.962
C00688=1082.108,397.618,-102.327,176.788,28.911,154.960
C00689=1082.102,397.371,-102.288,176.784,28.903,154.958
C00690=1082.095,397.125,-102.248,176.781,28.895,154.957
C00691=1082.088,396.878,-102.208,176.777,28.887,154.955
C00692=1082.082,396.631,-102.168,176.773,28.879,154.954
C00693=1082.076,396.385,-102.128,176.769,28.871,154.952
C00694=1082.069,396.139,-102.089,176.766,28.863,154.950
C00695=1082.063,395.891,-102.049,176.762,28.855,154.949
C00696=1082.056,395.645,-102.009,176.759,28.847,154.947
C00697=1082.050,395.398,-101.970,176.755,28.839,154.945
C00698=1082.043,395.152,-101.930,176.751,28.831,154.944
C00699=1082.037,394.905,-101.890,176.747,28.823,154.942
C00700=1082.031,394.658,-101.851,176.743,28.816,154.941
C00701=1082.024,394.411,-101.812,176.739,28.808,154.939
C00702=1082.018,394.165,-101.772,176.736,28.800,154.938
C00703=1082.012,393.918,-101.732,176.732,28.792,154.936
C00704=1082.004,393.671,-101.693,176.728,28.784,154.934
C00705=1081.998,393.424,-101.653,176.724,28.776,154.933
C00706=1081.991,393.178,-101.614,176.721,28.769,154.931
C00707=1081.985,392.931,-101.574,176.717,28.761,154.930
C00708=1081.978,392.684,-101.535,176.714,28.753,154.928
C00709=1081.972,392.437,-101.496,176.710,28.746,154.927
C00710=1081.965,392.191,-101.456,176.706,28.738,154.925
C00711=1081.959,391.944,-101.417,176.702,28.730,154.924
C00712=1081.954,391.697,-101.378,176.698,28.723,154.922
C00713=1081.947,391.450,-101.339,176.694,28.715,154.921
C00714=1081.940,391.204,-101.299,176.692,28.707,154.919
C00715=1081.934,390.957,-101.260,176.688,28.700,154.918
C00716=1081.927,390.710,-101.221,176.684,28.692,154.916
C00717=1081.920,390.463,-101.182,176.680,28.685,154.915
C00718=1081.914,390.216,-101.143,176.676,28.677,154.913
C00719=1081.907,389.969,-101.104,176.672,28.670,154.912
C00720=1081.901,389.723,-101.066,176.669,28.662,154.910
C00721=1081.895,389.476,-101.026,176.666,28.655,154.909
C00722=1081.888,389.229,-100.987,176.662,28.648,154.907
C00723=1081.881,388.982,-100.949,176.658,28.640,154.906
C00724=1081.874,388.736,-100.910,176.654,28.633,154.905
C00725=1081.869,388.489,-100.871,176.650,28.625,154.903
C00726=1081.862,388.242,-100.832,176.646,28.618,154.902
C00727=1081.855,387.996,-100.793,176.644,28.611,154.900
C00728=1081.849,387.748,-100.754,176.640,28.604,154.899
C00729=1081.843,387.502,-100.715,176.636,28.596,154.897
C00730=1081.836,387.255,-100.677,176.632,28.589,154.896
C00731=1081.830,387.008,-100.638,176.628,28.581,154.895
C00732=1081.823,386.762,-100.600,176.625,28.574,154.893
C00733=1081.817,386.515,-100.560,176.621,28.567,154.892
C00734=1081.811,386.268,-100.521,176.618,28.560,154.890
C00735=1081.805,386.021,-100.484,176.614,28.552,154.889
C00736=1081.798,385.774,-100.445,176.611,28.546,154.888
C00737=1081.792,385.545,-100.408,176.607,28.539,154.886
C00738=1081.786,385.317,-100.373,176.604,28.532,154.885
C00739=1081.780,385.087,-100.337,176.600,28.526,154.884
C00740=1081.775,384.859,-100.302,176.597,28.519,154.882
C00741=1081.768,384.630,-100.266,176.594,28.513,154.881
C00742=1081.762,384.402,-100.230,176.590,28.506,154.880
C00743=1081.757,384.172,-100.194,176.587,28.499,154.879
C00744=1081.751,383.943,-100.159,176.583,28.492,154.877
C00745=1081.745,383.696,-100.120,176.580,28.485,154.876
C00746=1081.739,383.450,-100.082,176.576,28.478,154.875
C00747=1081.732,383.203,-100.043,176.573,28.471,154.873
C00748=1081.726,382.956,-100.005,176.570,28.465,154.872
C00749=1081.720,382.708,-99.967,176.566,28.457,154.870
C00750=1081.714,382.462,-99.928,176.562,28.450,154.869
C00751=1081.707,382.215,-99.890,176.558,28.443,154.868
C00752=1081.701,381.969,-99.852,176.555,28.437,154.866
C00753=1081.695,381.721,-99.814,176.551,28.429,154.865
C00754=1081.689,381.475,-99.776,176.547,28.422,154.864
C00755=1081.682,381.227,-99.738,176.545,28.416,154.862
C00756=1081.675,380.981,-99.700,176.541,28.409,154.861
C00757=1081.669,380.734,-99.662,176.537,28.402,154.860
C00758=1081.662,380.486,-99.624,176.534,28.396,154.859
C00759=1081.656,380.240,-99.586,176.530,28.388,154.857
C00760=1081.650,379.993,-99.547,176.526,28.381,154.856
C00761=1081.644,379.746,-99.509,176.523,28.375,154.855
C00762=1081.637,379.499,-99.471,176.519,28.368,154.853
C00763=1081.631,379.252,-99.434,176.515,28.361,154.852
C00764=1081.625,379.005,-99.396,176.513,28.355,154.851
C00765=1081.618,378.758,-99.358,176.509,28.348,154.850
C00766=1081.612,378.511,-99.320,176.505,28.341,154.848
C00767=1081.606,378.264,-99.282,176.502,28.335,154.847
C00768=1081.600,378.017,-99.244,176.498,28.328,154.846
C00769=1081.593,377.770,-99.207,176.495,28.321,154.845
C00770=1081.587,377.523,-99.169,176.491,28.315,154.843
C00771=1081.581,377.276,-99.131,176.487,28.308,154.842
C00772=1081.574,377.029,-99.093,176.484,28.302,154.841
C00773=1081.568,376.782,-99.056,176.480,28.295,154.840
C00774=1081.561,376.535,-99.018,176.478,28.288,154.838
C00775=1081.555,376.288,-98.980,176.474,28.282,154.837
C00776=1081.550,376.041,-98.943,176.470,28.275,154.836
C00777=1081.543,375.794,-98.905,176.467,28.268,154.834
C00778=1081.537,375.547,-98.867,176.463,28.262,154.833
C00779=1081.531,375.300,-98.830,176.460,28.255,154.832
C00780=1081.525,375.054,-98.792,176.456,28.249,154.831
C00781=1081.519,374.806,-98.755,176.452,28.242,154.830
C00782=1081.513,374.559,-98.717,176.449,28.236,154.828
C00783=1081.506,374.312,-98.680,176.445,28.229,154.827
C00784=1081.500,374.064,-98.643,176.442,28.223,154.826
C00785=1081.494,373.818,-98.605,176.439,28.216,154.825
C00786=1081.487,373.571,-98.568,176.436,28.210,154.824
C00787=1081.481,373.323,-98.530,176.432,28.204,154.822
C00788=1081.474,373.077,-98.493,176.429,28.198,154.821
C00789=1081.469,372.829,-98.456,176.425,28.191,154.820
C00790=1081.462,372.582,-98.419,176.421,28.184,154.819
C00791=1081.456,372.335,-98.382,176.418,28.178,154.818
C00792=1081.449,372.088,-98.344,176.414,28.172,154.817
C00793=1081.444,371.874,-98.312,176.411,28.166,154.815
C00794=1081.438,371.659,-98.280,176.408,28.161,154.815
C00795=1081.433,371.444,-98.248,176.406,28.156,154.813
C00796=1081.427,371.229,-98.215,176.403,28.150,154.812
C00797=1081.423,371.015,-98.183,176.400,28.145,154.812
C00798=1081.417,370.800,-98.151,176.397,28.139,154.810
C00799=1081.412,370.585,-98.119,176.394,28.134,154.809
C00800=1081.406,370.371,-98.086,176.390,28.129,154.809
C00801=1081.400,370.124,-98.049,176.387,28.122,154.807
C00802=1081.394,369.877,-98.012,176.384,28.116,154.806
C00803=1081.388,369.630,-97.976,176.380,28.110,154.805
C00804=1081.381,369.383,-97.939,176.377,28.104,154.804
C00805=1081.375,369.135,-97.901,176.373,28.097,154.803
C00806=1081.368,368.888,-97.865,176.370,28.092,154.802
C00807=1081.363,368.641,-97.828,176.366,28.085,154.801
C00808=1081.357,368.394,-97.791,176.363,28.079,154.799
C00809=1081.350,368.147,-97.754,176.360,28.073,154.798
C00810=1081.344,367.900,-97.717,176.356,28.067,154.797
C00811=1081.338,367.653,-97.681,176.353,28.061,154.796
C00812=1081.332,367.406,-97.644,176.349,28.054,154.795
C00813=1081.325,367.158,-97.607,176.346,28.049,154.794
C00814=1081.319,366.911,-97.570,176.342,28.042,154.793
C00815=1081.314,366.663,-97.533,176.339,28.037,154.792
C00816=1081.307,366.416,-97.497,176.335,28.030,154.791
C00817=1081.301,366.169,-97.460,176.333,28.024,154.789
C00818=1081.295,365.922,-97.423,176.329,28.018,154.788
C00819=1081.289,365.675,-97.387,176.326,28.012,154.787
C00820=1081.283,365.428,-97.350,176.323,28.007,154.786
C00821=1081.277,365.181,-97.313,176.319,28.000,154.785
C00822=1081.271,364.933,-97.277,176.316,27.994,154.784
C00823=1081.264,364.686,-97.241,176.312,27.989,154.783
C00824=1081.258,364.439,-97.204,176.309,27.982,154.782
C00825=1081.252,364.192,-97.168,176.305,27.976,154.781
C00826=1081.246,363.944,-97.131,176.302,27.971,154.780
C00827=1081.240,363.697,-97.095,176.299,27.965,154.779
C00828=1081.234,363.450,-97.058,176.295,27.959,154.778
C00829=1081.227,363.203,-97.022,176.292,27.953,154.776
C00830=1081.221,362.956,-96.986,176.288,27.947,154.775
C00831=1081.215,362.708,-96.950,176.285,27.941,154.774
C00832=1081.209,362.461,-96.913,176.281,27.936,154.773
C00833=1081.202,362.214,-96.877,176.278,27.930,154.772
C00834=1081.196,361.967,-96.841,176.275,27.924,154.771
C00835=1081.190,361.720,-96.805,176.271,27.918,154.770
C00836=1081.184,361.472,-96.768,176.268,27.913,154.769
C00837=1081.178,361.225,-96.732,176.265,27.907,154.768
C00838=1081.172,360.978,-96.696,176.261,27.901,154.767
C00839=1081.166,360.730,-96.660,176.258,27.895,154.766
C00840=1081.160,360.483,-96.623,176.254,27.889,154.765
C00841=1081.154,360.235,-96.588,176.251,27.884,154.764
C00842=1081.147,359.988,-96.551,176.248,27.878,154.763
C00843=1081.141,359.740,-96.515,176.244,27.872,154.762
C00844=1081.135,359.494,-96.479,176.241,27.866,154.761
C00845=1081.129,359.246,-96.444,176.239,27.861,154.760
C00846=1081.123,358.999,-96.407,176.234,27.855,154.759
C00847=1081.117,358.752,-96.371,176.232,27.850,154.758
C00848=1081.110,358.505,-96.336,176.228,27.844,154.757
C00849=1081.100,358.091,-96.276,176.222,27.835,154.755
C00850=1081.090,357.678,-96.216,176.217,27.825,154.754
C00851=1081.079,357.265,-96.156,176.212,27.816,154.752
C00852=1081.069,356.851,-96.097,176.206,27.807,154.750
C00853=1081.063,356.604,-96.060,176.202,27.801,154.749
C00854=1081.057,356.357,-96.025,176.199,27.795,154.748
C00855=1081.051,356.110,-95.989,176.196,27.790,154.748
C00856=1081.045,355.862,-95.953,176.192,27.784,154.747
C00857=1081.038,355.615,-95.918,176.189,27.779,154.746
C00858=1081.033,355.368,-95.882,176.186,27.773,154.745
C00859=1081.027,355.121,-95.846,176.182,27.768,154.744
C00860=1081.021,354.873,-95.811,176.179,27.762,154.743
C00861=1081.015,354.625,-95.775,176.176,27.757,154.742
C00862=1081.008,354.378,-95.740,176.172,27.751,154.741
C00863=1081.002,354.131,-95.704,176.169,27.746,154.740
C00864=1080.996,353.883,-95.669,176.166,27.740,154.739
C00865=1080.990,353.636,-95.633,176.163,27.735,154.738
C00866=1080.984,353.389,-95.598,176.159,27.730,154.737
C00867=1080.978,353.141,-95.562,176.156,27.724,154.736
C00868=1080.972,352.894,-95.527,176.153,27.719,154.735
C00869=1080.966,352.646,-95.491,176.149,27.713,154.734
C00870=1080.960,352.399,-95.456,176.146,27.708,154.733
C00871=1080.954,352.152,-95.421,176.143,27.702,154.732
C00872=1080.947,351.904,-95.385,176.140,27.697,154.731
C00873=1080.942,351.657,-95.350,176.136,27.692,154.730
C00874=1080.936,351.409,-95.315,176.133,27.686,154.729
C00875=1080.929,351.162,-95.280,176.130,27.681,154.729
C00876=1080.923,350.914,-95.244,176.127,27.676,154.728
C00877=1080.917,350.667,-95.209,176.123,27.671,154.727
C00878=1080.911,350.420,-95.174,176.120,27.665,154.726
C00879=1080.905,350.172,-95.139,176.117,27.660,154.725
C00880=1080.899,349.925,-95.104,176.114,27.654,154.724
C00881=1080.893,349.677,-95.068,176.110,27.649,154.723
C00882=1080.887,349.430,-95.033,176.107,27.644,154.722
C00883=1080.881,349.182,-94.998,176.104,27.639,154.721
C00884=1080.874,348.935,-94.963,176.101,27.633,154.720
C00885=1080.869,348.688,-94.928,176.097,27.628,154.719
C00886=1080.863,348.440,-94.893,176.094,27.623,154.718
C00887=1080.857,348.193,-94.858,176.091,27.618,154.718
C00888=1080.851,347.945,-94.824,176.088,27.613,154.717
C00889=1080.845,347.697,-94.788,176.085,27.608,154.716
C00890=1080.839,347.450,-94.754,176.081,27.602,154.715
C00891=1080.832,347.202,-94.719,176.078,27.597,154.714
C00892=1080.827,346.955,-94.684,176.075,27.592,154.713
C00893=1080.820,346.707,-94.649,176.072,27.586,154.712
C00894=1080.815,346.460,-94.614,176.069,27.582,154.711
C00895=1080.808,346.212,-94.579,176.065,27.576,154.711
C00896=1080.803,345.965,-94.545,176.062,27.571,154.710
C00897=1080.796,345.717,-94.509,176.059,27.566,154.709
C00898=1080.790,345.469,-94.475,176.056,27.561,154.708
C00899=1080.784,345.223,-94.440,176.053,27.556,154.707
C00900=1080.778,344.975,-94.405,176.050,27.551,154.706
C00901=1080.768,344.565,-94.348,176.044,27.542,154.705
C00902=1080.759,344.155,-94.290,176.039,27.534,154.703
C00903=1080.749,343.744,-94.233,176.034,27.525,154.702
C00904=1080.739,343.334,-94.176,176.028,27.517,154.701
C00905=1080.732,343.086,-94.142,176.025,27.512,154.700
C00906=1080.726,342.839,-94.108,176.022,27.507,154.699
C00907=1080.719,342.592,-94.072,176.018,27.502,154.698
C00908=1080.714,342.344,-94.038,176.015,27.497,154.697
C00909=1080.708,342.096,-94.003,176.012,27.492,154.696
C00910=1080.702,341.849,-93.969,176.009,27.487,154.696
C00911=1080.696,341.602,-93.935,176.006,27.482,154.695
C00912=1080.690,341.354,-93.901,176.003,27.477,154.694
C00913=1080.685,341.106,-93.866,176.000,27.472,154.693
C00914=1080.678,340.859,-93.831,175.996,27.467,154.692
C00915=1080.672,340.611,-93.797,175.993,27.462,154.691
C00916=1080.666,340.364,-93.763,175.990,27.457,154.691
C00917=1080.660,340.116,-93.728,175.986,27.452,154.690
C00918=1080.654,339.869,-93.694,175.983,27.447,154.689
C00919=1080.647,339.621,-93.660,175.980,27.442,154.688
C00920=1080.642,339.373,-93.625,175.977,27.437,154.687
C00921=1080.636,339.126,-93.591,175.974,27.432,154.686
C00922=1080.630,338.877,-93.558,175.971,27.427,154.686
C00923=1080.624,338.630,-93.524,175.967,27.422,154.685
C00924=1080.618,338.383,-93.490,175.964,27.417,154.684
C00925=1080.612,338.135,-93.455,175.961,27.412,154.683
C00926=1080.606,337.888,-93.421,175.958,27.408,154.682
C00927=1080.600,337.640,-93.387,175.955,27.403,154.682
C00928=1080.594,337.392,-93.353,175.952,27.398,154.681
C00929=1080.588,337.144,-93.319,175.949,27.393,154.680
C00930=1080.582,336.897,-93.285,175.946,27.388,154.679
C00931=1080.576,336.649,-93.251,175.943,27.383,154.678
C00932=1080.570,336.402,-93.217,175.940,27.379,154.678
C00933=1080.564,336.154,-93.183,175.937,27.374,154.677
C00934=1080.559,335.907,-93.149,175.933,27.369,154.676
C00935=1080.552,335.659,-93.115,175.929,27.364,154.675
C00936=1080.546,335.412,-93.081,175.926,27.359,154.674
C00937=1080.540,335.164,-93.048,175.923,27.355,154.674
C00938=1080.534,334.916,-93.014,175.920,27.350,154.673
C00939=1080.528,334.668,-92.980,175.917,27.345,154.672
C00940=1080.522,334.421,-92.946,175.914,27.340,154.671
C00941=1080.516,334.173,-92.912,175.911,27.336,154.671
C00942=1080.511,333.925,-92.879,175.908,27.331,154.670
C00943=1080.504,333.677,-92.844,175.905,27.326,154.669
C00944=1080.498,333.430,-92.812,175.902,27.321,154.668
C00945=1080.492,333.183,-92.778,175.899,27.317,154.667
C00946=1080.487,332.935,-92.744,175.896,27.312,154.667
C00947=1080.481,332.687,-92.710,175.893,27.307,154.666
C00948=1080.475,332.439,-92.677,175.890,27.302,154.665
C00949=1080.469,332.192,-92.643,175.886,27.298,154.664
C00950=1080.463,331.944,-92.609,175.883,27.293,154.664
C00951=1080.456,331.697,-92.576,175.880,27.288,154.663
C00952=1080.451,331.449,-92.542,175.877,27.283,154.662
C00953=1080.440,331.033,-92.486,175.872,27.276,154.661
C00954=1080.430,330.618,-92.430,175.866,27.268,154.660
C00955=1080.420,330.202,-92.374,175.862,27.261,154.658
C00956=1080.410,329.786,-92.318,175.856,27.253,154.657
C00957=1080.404,329.539,-92.285,175.853,27.248,154.656
C00958=1080.397,329.290,-92.252,175.850,27.243,154.656
C00959=1080.391,329.043,-92.218,175.847,27.239,154.655
C00960=1080.385,328.795,-92.185,175.844,27.234,154.654
C00961=1080.379,328.548,-92.152,175.841,27.230,154.653
C00962=1080.373,328.300,-92.119,175.838,27.225,154.653
C00963=1080.367,328.052,-92.086,175.835,27.221,154.652
C00964=1080.361,327.805,-92.052,175.832,27.216,154.651
C00965=1080.354,327.557,-92.019,175.828,27.212,154.651
C00966=1080.349,327.309,-91.986,175.825,27.207,154.650
C00967=1080.343,327.061,-91.953,175.822,27.203,154.649
C00968=1080.337,326.813,-91.919,175.819,27.198,154.648
C00969=1080.331,326.566,-91.887,175.816,27.194,154.648
C00970=1080.325,326.318,-91.853,175.813,27.189,154.647
C00971=1080.319,326.070,-91.821,175.810,27.185,154.646
C00972=1080.313,325.822,-91.787,175.807,27.180,154.645
C00973=1080.307,325.575,-91.755,175.804,27.175,154.645
C00974=1080.301,325.327,-91.722,175.801,27.171,154.644
C00975=1080.295,325.079,-91.688,175.797,27.166,154.643
C00976=1080.289,324.832,-91.656,175.794,27.162,154.643
C00977=1080.283,324.584,-91.622,175.792,27.158,154.642
C00978=1080.277,324.336,-91.590,175.789,27.153,154.641
C00979=1080.271,324.088,-91.556,175.786,27.149,154.641
C00980=1080.265,323.841,-91.524,175.783,27.144,154.640
C00981=1080.259,323.593,-91.491,175.780,27.140,154.639
C00982=1080.253,323.345,-91.457,175.777,27.135,154.638
C00983=1080.247,323.097,-91.425,175.774,27.131,154.638
C00984=1080.242,322.849,-91.392,175.771,27.126,154.637
C00985=1080.236,322.601,-91.359,175.767,27.122,154.636
C00986=1080.229,322.354,-91.327,175.764,27.117,154.636
C00987=1080.224,322.106,-91.293,175.761,27.113,154.635
C00988=1080.218,321.858,-91.261,175.758,27.108,154.634
C00989=1080.212,321.611,-91.229,175.755,27.104,154.634
C00990=1080.206,321.363,-91.196,175.753,27.100,154.633
C00991=1080.200,321.115,-91.163,175.750,27.095,154.632
C00992=1080.194,320.867,-91.131,175.747,27.091,154.631
C00993=1080.189,320.619,-91.097,175.744,27.086,154.631
C00994=1080.182,320.372,-91.065,175.740,27.082,154.630
C00995=1080.176,320.123,-91.033,175.737,27.077,154.629
C00996=1080.171,319.876,-91.000,175.734,27.073,154.629
C00997=1080.165,319.629,-90.967,175.731,27.068,154.628
C00998=1080.159,319.380,-90.935,175.728,27.064,154.627
C00999=1080.154,319.132,-90.902,175.725,27.059,154.627
C01000=1080.148,318.884,-90.870,175.723,27.055,154.626
C01001=1080.142,318.637,-90.837,175.720,27.051,154.625
C01002=1080.137,318.389,-90.805,175.717,27.046,154.624
C01003=1080.130,318.141,-90.772,175.714,27.042,154.624
C01004=1080.124,317.894,-90.739,175.710,27.038,154.623
C01005=1080.120,317.682,-90.712,175.708,27.034,154.622
C01006=1080.115,317.471,-90.684,175.706,27.030,154.622
C01007=1080.109,317.260,-90.657,175.703,27.026,154.621
C01008=1080.105,317.049,-90.629,175.701,27.022,154.621
C01009=1080.100,316.839,-90.601,175.698,27.019,154.620
C01010=1080.095,316.626,-90.574,175.695,27.015,154.620
C01011=1080.090,316.416,-90.546,175.693,27.011,154.619
C01012=1080.086,316.205,-90.518,175.691,27.008,154.618
C01013=1080.080,315.957,-90.486,175.687,27.003,154.618
C01014=1080.073,315.709,-90.454,175.684,26.999,154.617
C01015=1080.068,315.461,-90.422,175.681,26.994,154.616
C01016=1080.062,315.214,-90.389,175.678,26.990,154.616
C01017=1080.056,314.965,-90.357,175.676,26.986,154.615
C01018=1080.051,314.718,-90.325,175.673,26.982,154.614
C01019=1080.045,314.470,-90.293,175.670,26.977,154.614
C01020=1080.039,314.222,-90.260,175.667,26.973,154.613
C01021=1080.032,313.974,-90.229,175.663,26.969,154.612
C01022=1080.026,313.726,-90.197,175.660,26.965,154.612
C01023=1080.021,313.478,-90.165,175.658,26.961,154.611
C01024=1080.014,313.231,-90.132,175.655,26.956,154.610
C01025=1080.008,312.983,-90.100,175.652,26.952,154.610
C01026=1080.002,312.734,-90.068,175.649,26.948,154.609
C01027=1079.996,312.487,-90.037,175.646,26.944,154.609
C01028=1079.990,312.239,-90.005,175.643,26.940,154.608
C01029=1079.984,311.991,-89.973,175.640,26.936,154.607
C01030=1079.979,311.743,-89.941,175.637,26.931,154.607
C01031=1079.972,311.496,-89.909,175.634,26.927,154.606
C01032=1079.966,311.248,-89.877,175.631,26.923,154.605
C01033=1079.960,311.000,-89.846,175.628,26.919,154.605
C01034=1079.954,310.752,-89.814,175.625,26.915,154.604
C01035=1079.948,310.504,-89.782,175.622,26.911,154.604
C01036=1079.942,310.257,-89.751,175.619,26.906,154.603
C01037=1079.936,310.008,-89.719,175.616,26.902,154.602
C01038=1079.930,309.760,-89.686,175.613,26.898,154.602
C01039=1079.925,309.513,-89.655,175.610,26.894,154.601
C01040=1079.918,309.265,-89.623,175.608,26.890,154.600
C01041=1079.913,309.017,-89.592,175.605,26.886,154.600
C01042=1079.907,308.769,-89.560,175.602,26.881,154.599
C01043=1079.900,308.521,-89.528,175.598,26.877,154.599
C01044=1079.895,308.274,-89.497,175.595,26.873,154.598
C01045=1079.889,308.025,-89.465,175.593,26.869,154.597
C01046=1079.884,307.777,-89.434,175.590,26.865,154.597
C01047=1079.877,307.529,-89.402,175.587,26.860,154.596
C01048=1079.872,307.282,-89.371,175.584,26.856,154.595
C01049=1079.866,307.034,-89.339,175.581,26.852,154.595
C01050=1079.859,306.786,-89.307,175.578,26.848,154.594
C01051=1079.854,306.538,-89.276,175.575,26.844,154.594
C01052=1079.848,306.290,-89.244,175.572,26.840,154.593
C01053=1079.842,306.042,-89.213,175.569,26.836,154.592
C01054=1079.836,305.795,-89.181,175.567,26.832,154.592
C01055=1079.830,305.546,-89.149,175.564,26.828,154.591
C01056=1079.824,305.299,-89.119,175.561,26.823,154.590
C01057=1079.818,305.050,-89.087,175.557,26.819,154.590
C01058=1079.813,304.803,-89.055,175.554,26.815,154.589
C01059=1079.807,304.554,-89.025,175.552,26.811,154.589
C01060=1079.801,304.307,-88.993,175.549,26.807,154.588
C01061=1079.791,303.888,-88.940,175.544,26.800,154.587
C01062=1079.782,303.469,-88.887,175.539,26.793,154.586
C01063=1079.771,303.050,-88.834,175.534,26.786,154.585
C01064=1079.762,302.631,-88.781,175.530,26.780,154.584
C01065=1079.756,302.382,-88.750,175.527,26.775,154.583
C01066=1079.750,302.135,-88.719,175.524,26.771,154.583
C01067=1079.744,301.886,-88.688,175.521,26.767,154.582
C01068=1079.738,301.639,-88.656,175.518,26.763,154.581
C01069=1079.733,301.391,-88.626,175.515,26.759,154.581
C01070=1079.727,301.143,-88.594,175.512,26.754,154.580
C01071=1079.721,300.895,-88.563,175.509,26.751,154.580
C01072=1079.716,300.647,-88.531,175.507,26.747,154.579
C01073=1079.710,300.399,-88.501,175.504,26.742,154.578
C01074=1079.705,300.151,-88.470,175.501,26.738,154.578
C01075=1079.698,299.903,-88.439,175.497,26.734,154.577
C01076=1079.693,299.655,-88.408,175.495,26.730,154.577
C01077=1079.687,299.407,-88.377,175.492,26.726,154.576
C01078=1079.682,299.159,-88.345,175.489,26.722,154.575
C01079=1079.676,298.911,-88.315,175.487,26.718,154.575
C01080=1079.670,298.664,-88.283,175.484,26.713,154.574
C01081=1079.664,298.415,-88.253,175.481,26.710,154.574
C01082=1079.659,298.167,-88.222,175.478,26.706,154.573
C01083=1079.653,297.919,-88.191,175.475,26.701,154.572
C01084=1079.648,297.672,-88.160,175.472,26.697,154.572
C01085=1079.641,297.423,-88.129,175.469,26.693,154.571
C01086=1079.635,297.176,-88.099,175.467,26.690,154.571
C01087=1079.630,296.927,-88.068,175.464,26.685,154.570
C01088=1079.624,296.679,-88.037,175.461,26.681,154.569
C01089=1079.618,296.432,-88.006,175.458,26.677,154.569
C01090=1079.612,296.184,-87.976,175.455,26.674,154.568
C01091=1079.606,295.935,-87.944,175.452,26.670,154.568
C01092=1079.600,295.687,-87.914,175.450,26.666,154.567
C01093=1079.595,295.439,-87.884,175.447,26.662,154.566
C01094=1079.589,295.192,-87.853,175.444,26.658,154.566
C01095=1079.583,294.943,-87.822,175.441,26.654,154.565
C01096=1079.577,294.695,-87.792,175.438,26.650,154.565
C01097=1079.572,294.447,-87.761,175.435,26.646,154.564
C01098=1079.566,294.199,-87.731,175.433,26.642,154.564
C01099=1079.559,293.951,-87.700,175.430,26.638,154.563
C01100=1079.553,293.703,-87.670,175.427,26.634,154.562
C01101=1079.548,293.455,-87.639,175.425,26.630,154.562
C01102=1079.543,293.207,-87.608,175.421,26.626,154.561
C01103=1079.537,292.959,-87.578,175.418,26.622,154.561
C01104=1079.530,292.711,-87.547,175.416,26.618,154.560
C01105=1079.525,292.463,-87.517,175.413,26.615,154.560
C01106=1079.519,292.215,-87.487,175.410,26.610,154.559
C01107=1079.513,291.967,-87.456,175.408,26.607,154.558
C01108=1079.507,291.719,-87.426,175.404,26.603,154.558
C01109=1079.501,291.471,-87.395,175.401,26.598,154.557
C01110=1079.496,291.223,-87.364,175.399,26.595,154.557
C01111=1079.490,290.974,-87.335,175.396,26.591,154.556
C01112=1079.484,290.726,-87.304,175.393,26.587,154.556
C01113=1079.474,290.322,-87.255,175.388,26.581,154.555
C01114=1079.465,289.917,-87.205,175.385,26.574,154.554
C01115=1079.455,289.512,-87.156,175.380,26.568,154.553
C01116=1079.446,289.108,-87.107,175.375,26.561,154.552
C01117=1079.440,288.859,-87.077,175.372,26.558,154.551
C01118=1079.434,288.612,-87.046,175.369,26.554,154.551
C01119=1079.428,288.363,-87.017,175.367,26.550,154.550
C01120=1079.423,288.115,-86.986,175.364,26.546,154.550
C01121=1079.417,287.868,-86.956,175.361,26.542,154.549
C01122=1079.411,287.619,-86.926,175.358,26.538,154.549
C01123=1079.405,287.372,-86.897,175.355,26.535,154.548
C01124=1079.399,287.123,-86.867,175.353,26.531,154.548
C01125=1079.393,286.875,-86.836,175.350,26.527,154.547
C01126=1079.387,286.627,-86.806,175.347,26.523,154.546
C01127=1079.381,286.378,-86.776,175.344,26.519,154.546
C01128=1079.376,286.131,-86.746,175.341,26.515,154.545
C01129=1079.370,285.882,-86.716,175.339,26.512,154.545
C01130=1079.364,285.635,-86.687,175.336,26.508,154.544
C01131=1079.358,285.386,-86.657,175.333,26.504,154.544
C01132=1079.352,285.138,-86.627,175.331,26.500,154.543
C01133=1079.347,284.890,-86.597,175.327,26.496,154.543
C01134=1079.341,284.642,-86.567,175.325,26.492,154.542
C01135=1079.335,284.394,-86.538,175.322,26.488,154.541
C01136=1079.329,284.146,-86.507,175.320,26.485,154.541
C01137=1079.323,283.898,-86.478,175.317,26.481,154.540
C01138=1079.318,283.649,-86.448,175.314,26.477,154.540
C01139=1079.312,283.401,-86.418,175.312,26.473,154.539
C01140=1079.306,283.153,-86.389,175.308,26.469,154.539
C01141=1079.300,282.905,-86.359,175.306,26.466,154.538
C01142=1079.294,282.657,-86.329,175.303,26.462,154.538
C01143=1079.289,282.409,-86.299,175.300,26.457,154.537
C01144=1079.283,282.160,-86.269,175.298,26.454,154.536
C01145=1079.277,281.913,-86.240,175.295,26.450,154.536
C01146=1079.271,281.664,-86.210,175.292,26.446,154.535
C01147=1079.266,281.416,-86.180,175.289,26.443,154.535
C01148=1079.260,281.168,-86.150,175.287,26.439,154.534
C01149=1079.254,280.920,-86.121,175.284,26.435,154.534
C01150=1079.249,280.672,-86.092,175.282,26.431,154.533
C01151=1079.243,280.424,-86.062,175.279,26.427,154.533
C01152=1079.237,280.175,-86.033,175.275,26.423,154.532
C01153=1079.232,279.927,-86.003,175.273,26.420,154.532
C01154=1079.225,279.680,-85.974,175.270,26.416,154.531
C01155=1079.219,279.431,-85.944,175.268,26.412,154.531
C01156=1079.213,279.183,-85.915,175.265,26.409,154.530
C01157=1079.208,278.935,-85.885,175.263,26.405,154.529
C01158=1079.202,278.686,-85.856,175.259,26.401,154.529
C01159=1079.196,278.438,-85.827,175.257,26.397,154.528
C01160=1079.190,278.189,-85.797,175.254,26.393,154.528
C01161=1079.184,277.941,-85.768,175.251,26.389,154.527
C01162=1079.179,277.693,-85.738,175.249,26.386,154.527
C01163=1079.173,277.445,-85.710,175.246,26.382,154.526
C01164=1079.168,277.197,-85.680,175.243,26.378,154.526
C01165=1079.158,276.802,-85.633,175.239,26.372,154.525
C01166=1079.149,276.407,-85.586,175.235,26.367,154.524
C01167=1079.140,276.012,-85.540,175.230,26.360,154.523
C01168=1079.130,275.618,-85.493,175.226,26.354,154.522
C01169=1079.125,275.369,-85.464,175.224,26.350,154.522
C01170=1079.118,275.121,-85.435,175.220,26.346,154.521
C01171=1079.114,274.873,-85.406,175.218,26.343,154.521
C01172=1079.107,274.625,-85.377,175.215,26.339,154.520
C01173=1079.101,274.376,-85.348,175.213,26.335,154.520
C01174=1079.096,274.128,-85.318,175.210,26.332,154.519
C01175=1079.089,273.880,-85.289,175.207,26.328,154.519
C01176=1079.085,273.632,-85.260,175.204,26.324,154.518
C01177=1079.079,273.383,-85.232,175.202,26.321,154.518
C01178=1079.072,273.135,-85.203,175.199,26.317,154.517
C01179=1079.067,272.887,-85.173,175.197,26.313,154.517
C01180=1079.061,272.639,-85.144,175.194,26.309,154.516
C01181=1079.055,272.391,-85.116,175.191,26.306,154.516
C01182=1079.050,272.142,-85.086,175.188,26.302,154.515
C01183=1079.043,271.894,-85.057,175.186,26.298,154.514
C01184=1079.038,271.645,-85.029,175.183,26.294,154.514
C01185=1079.033,271.398,-85.000,175.181,26.291,154.513
C01186=1079.026,271.149,-84.971,175.178,26.287,154.513
C01187=1079.020,270.901,-84.942,175.175,26.283,154.512
C01188=1079.014,270.653,-84.913,175.172,26.279,154.512
C01189=1079.009,270.405,-84.884,175.170,26.276,154.511
C01190=1079.003,270.156,-84.856,175.167,26.272,154.511
C01191=1078.997,269.908,-84.827,175.165,26.268,154.510
C01192=1078.991,269.659,-84.798,175.162,26.265,154.510
C01193=1078.986,269.411,-84.769,175.159,26.261,154.509
C01194=1078.980,269.163,-84.740,175.156,26.257,154.509
C01195=1078.974,268.915,-84.712,175.154,26.254,154.508
C01196=1078.968,268.667,-84.683,175.151,26.250,154.508
C01197=1078.962,268.418,-84.655,175.149,26.246,154.507
C01198=1078.957,268.170,-84.625,175.147,26.243,154.507
C01199=1078.951,267.921,-84.597,175.143,26.239,154.506
C01200=1078.945,267.674,-84.568,175.141,26.236,154.506
C01201=1078.939,267.425,-84.540,175.138,26.232,154.505
C01202=1078.933,267.176,-84.512,175.136,26.228,154.505
C01203=1078.928,266.929,-84.483,175.133,26.224,154.504
C01204=1078.922,266.680,-84.455,175.130,26.221,154.504
C01205=1078.916,266.432,-84.425,175.127,26.217,154.503
C01206=1078.911,266.184,-84.397,175.125,26.213,154.503
C01207=1078.905,265.935,-84.369,175.122,26.209,154.502
C01208=1078.899,265.687,-84.340,175.120,26.206,154.502
C01209=1078.893,265.439,-84.312,175.117,26.202,154.501
C01210=1078.888,265.190,-84.283,175.114,26.198,154.501
C01211=1078.882,264.942,-84.255,175.112,26.195,154.500
C01212=1078.876,264.694,-84.226,175.109,26.191,154.499
C01213=1078.870,264.445,-84.198,175.107,26.187,154.499
C01214=1078.864,264.198,-84.169,175.104,26.183,154.498
C01215=1078.858,263.949,-84.141,175.102,26.180,154.498
C01216=1078.853,263.701,-84.113,175.098,26.176,154.498
C01217=1078.843,263.309,-84.068,175.095,26.171,154.497
C01218=1078.834,262.917,-84.023,175.091,26.165,154.496
C01219=1078.825,262.525,-83.979,175.086,26.159,154.495
C01220=1078.815,262.133,-83.935,175.083,26.154,154.494
C01221=1078.810,261.885,-83.906,175.079,26.150,154.494
C01222=1078.804,261.636,-83.878,175.077,26.146,154.493
C01223=1078.798,261.388,-83.850,175.074,26.143,154.493
C01224=1078.792,261.140,-83.822,175.072,26.139,154.492
C01225=1078.786,260.891,-83.794,175.070,26.136,154.492
C01226=1078.780,260.643,-83.766,175.066,26.132,154.491
C01227=1078.774,260.394,-83.738,175.064,26.128,154.491
C01228=1078.768,260.146,-83.709,175.061,26.124,154.490
C01229=1078.762,259.898,-83.682,175.059,26.121,154.490
C01230=1078.756,259.649,-83.654,175.056,26.117,154.489
C01231=1078.751,259.401,-83.626,175.054,26.114,154.489
C01232=1078.745,259.152,-83.597,175.051,26.110,154.488
C01233=1078.739,258.905,-83.570,175.048,26.106,154.488
C01234=1078.733,258.656,-83.542,175.046,26.103,154.487
C01235=1078.728,258.408,-83.514,175.043,26.099,154.487
C01236=1078.722,258.159,-83.485,175.041,26.096,154.486
C01237=1078.716,257.911,-83.458,175.039,26.092,154.486
C01238=1078.710,257.663,-83.430,175.035,26.088,154.485
C01239=1078.705,257.414,-83.403,175.033,26.085,154.485
C01240=1078.698,257.165,-83.375,175.030,26.081,154.485
C01241=1078.693,256.917,-83.347,175.028,26.078,154.484
C01242=1078.687,256.669,-83.319,175.026,26.074,154.483
C01243=1078.681,256.421,-83.291,175.023,26.070,154.483
C01244=1078.675,256.172,-83.263,175.020,26.067,154.482
C01245=1078.670,255.924,-83.236,175.018,26.063,154.482
C01246=1078.664,255.675,-83.207,175.015,26.060,154.482
C01247=1078.658,255.427,-83.180,175.013,26.056,154.481
C01248=1078.652,255.179,-83.152,175.010,26.052,154.480
C01249=1078.646,254.930,-83.124,175.007,26.049,154.480
C01250=1078.641,254.682,-83.097,175.005,26.045,154.479
C01251=1078.635,254.433,-83.069,175.002,26.041,154.479
C01252=1078.629,254.185,-83.041,175.000,26.038,154.479
C01253=1078.624,253.937,-83.014,174.998,26.034,154.478
C01254=1078.618,253.688,-82.986,174.995,26.030,154.477
C01255=1078.612,253.440,-82.958,174.992,26.027,154.477
C01256=1078.606,253.191,-82.931,174.989,26.023,154.476
C01257=1078.601,252.943,-82.903,174.987,26.019,154.476
C01258=1078.595,252.695,-82.875,174.985,26.016,154.475
C01259=1078.589,252.446,-82.848,174.982,26.012,154.475
C01260=1078.584,252.198,-82.820,174.980,26.009,154.474
C01261=1078.578,251.949,-82.793,174.977,26.005,154.474
C01262=1078.572,251.701,-82.765,174.974,26.001,154.473
C01263=1078.567,251.452,-82.737,174.972,25.998,154.473
C01264=1078.561,251.204,-82.710,174.970,25.994,154.472
C01265=1078.555,250.955,-82.682,174.967,25.990,154.472
C01266=1078.550,250.707,-82.655,174.965,25.987,154.471
C01267=1078.544,250.459,-82.627,174.962,25.983,154.471
C01268=1078.538,250.210,-82.600,174.959,25.980,154.470
C01269=1078.529,249.815,-82.556,174.956,25.974,154.470
C01270=1078.520,249.421,-82.513,174.952,25.968,154.469
C01271=1078.511,249.026,-82.470,174.948,25.962,154.468
C01272=1078.502,248.632,-82.426,174.944,25.956,154.467
C01273=1078.497,248.384,-82.398,174.942,25.953,154.467
C01274=1078.491,248.135,-82.371,174.938,25.949,154.466
C01275=1078.485,247.887,-82.343,174.936,25.945,154.466
C01276=1078.480,247.638,-82.317,174.934,25.942,154.465
C01277=1078.474,247.390,-82.289,174.931,25.938,154.465
C01278=1078.468,247.142,-82.262,174.929,25.934,154.464
C01279=1078.463,246.892,-82.234,174.927,25.931,154.464
C01280=1078.457,246.644,-82.208,174.924,25.927,154.463
C01281=1078.452,246.396,-82.180,174.921,25.924,154.463
C01282=1078.446,246.148,-82.153,174.919,25.920,154.462
C01283=1078.440,245.899,-82.126,174.916,25.916,154.462
C01284=1078.434,245.650,-82.099,174.914,25.912,154.461
C01285=1078.428,245.402,-82.072,174.912,25.909,154.461
C01286=1078.423,245.154,-82.045,174.910,25.906,154.460
C01287=1078.418,244.905,-82.018,174.906,25.902,154.460
C01288=1078.411,244.656,-81.991,174.904,25.898,154.459
C01289=1078.405,244.408,-81.964,174.902,25.895,154.459
C01290=1078.400,244.160,-81.936,174.899,25.891,154.458
C01291=1078.394,243.911,-81.909,174.897,25.887,154.458
C01292=1078.389,243.663,-81.883,174.895,25.884,154.457
C01293=1078.383,243.414,-81.855,174.892,25.880,154.457
C01294=1078.377,243.165,-81.829,174.889,25.876,154.456
C01295=1078.371,242.917,-81.802,174.887,25.873,154.456
C01296=1078.366,242.669,-81.775,174.885,25.870,154.455
C01297=1078.361,242.420,-81.748,174.882,25.866,154.455
C01298=1078.355,242.171,-81.721,174.880,25.862,154.454
C01299=1078.348,241.922,-81.694,174.878,25.858,154.454
C01300=1078.343,241.674,-81.668,174.874,25.855,154.453
C01301=1078.337,241.426,-81.641,174.872,25.851,154.453
C01302=1078.331,241.177,-81.614,174.870,25.848,154.452
C01303=1078.325,240.929,-81.588,174.868,25.844,154.452
C01304=1078.320,240.680,-81.561,174.865,25.841,154.451
C01305=1078.314,240.431,-81.534,174.863,25.837,154.451
C01306=1078.308,240.183,-81.507,174.860,25.834,154.450
C01307=1078.302,239.935,-81.480,174.857,25.830,154.450
C01308=1078.297,239.686,-81.454,174.855,25.826,154.449
C01309=1078.291,239.438,-81.427,174.853,25.823,154.449
C01310=1078.285,239.189,-81.400,174.851,25.819,154.448
C01311=1078.279,238.941,-81.374,174.848,25.815,154.448
C01312=1078.273,238.692,-81.347,174.845,25.812,154.447
C01313=1078.267,238.444,-81.320,174.843,25.809,154.447
C01314=1078.262,238.195,-81.294,174.841,25.805,154.446
C01315=1078.256,237.946,-81.267,174.838,25.801,154.446
C01316=1078.250,237.698,-81.241,174.836,25.798,154.445
C01317=1078.244,237.450,-81.214,174.834,25.794,154.445
C01318=1078.239,237.201,-81.187,174.831,25.791,154.444
C01319=1078.233,236.953,-81.161,174.828,25.787,154.444
C01320=1078.227,236.704,-81.135,174.826,25.784,154.444
C01321=1078.218,236.303,-81.091,174.823,25.778,154.443
C01322=1078.209,235.901,-81.048,174.819,25.772,154.442
C01323=1078.200,235.500,-81.007,174.814,25.766,154.441
C01324=1078.191,235.099,-80.963,174.811,25.760,154.440
C01325=1078.185,234.850,-80.937,174.808,25.757,154.440
C01326=1078.180,234.602,-80.911,174.806,25.753,154.439
C01327=1078.174,234.353,-80.884,174.803,25.749,154.439
C01328=1078.168,234.104,-80.858,174.801,25.745,154.438
C01329=1078.162,233.856,-80.832,174.799,25.742,154.438
C01330=1078.156,233.608,-80.805,174.797,25.739,154.437
C01331=1078.151,233.359,-80.779,174.794,25.735,154.437
C01332=1078.145,233.111,-80.753,174.792,25.731,154.436
C01333=1078.139,232.862,-80.727,174.789,25.728,154.436
C01334=1078.134,232.613,-80.700,174.787,25.724,154.435
C01335=1078.128,232.364,-80.674,174.785,25.721,154.435
C01336=1078.122,232.116,-80.648,174.782,25.717,154.434
C01337=1078.116,231.868,-80.621,174.780,25.714,154.434
C01338=1078.110,231.619,-80.596,174.778,25.710,154.433
C01339=1078.105,231.371,-80.569,174.775,25.706,154.433
C01340=1078.099,231.122,-80.543,174.772,25.702,154.432
C01341=1078.094,230.873,-80.517,174.770,25.699,154.432
C01342=1078.088,230.624,-80.490,174.768,25.696,154.431
C01343=1078.082,230.376,-80.465,174.766,25.692,154.431
C01344=1078.076,230.127,-80.438,174.764,25.688,154.430
C01345=1078.071,229.879,-80.413,174.761,25.685,154.430
C01346=1078.065,229.631,-80.386,174.758,25.681,154.430
C01347=1078.059,229.382,-80.361,174.756,25.678,154.429
C01348=1078.054,229.133,-80.335,174.754,25.674,154.428
C01349=1078.048,228.885,-80.308,174.752,25.671,154.428
C01350=1078.042,228.636,-80.283,174.749,25.667,154.428
C01351=1078.036,228.387,-80.257,174.747,25.663,154.427
C01352=1078.030,228.139,-80.230,174.745,25.660,154.427
C01353=1078.024,227.890,-80.205,174.742,25.657,154.426
C01354=1078.019,227.641,-80.179,174.740,25.653,154.426
C01355=1078.012,227.393,-80.153,174.737,25.649,154.425
C01356=1078.007,227.144,-80.127,174.735,25.645,154.425
C01357=1078.002,226.896,-80.102,174.733,25.642,154.424
C01358=1077.996,226.647,-80.076,174.731,25.639,154.424
C01359=1077.990,226.399,-80.050,174.728,25.635,154.423
C01360=1077.985,226.150,-80.024,174.725,25.631,154.423
C01361=1077.978,225.901,-79.998,174.723,25.628,154.422
C01362=1077.973,225.652,-79.972,174.721,25.624,154.422
C01363=1077.967,225.403,-79.947,174.719,25.621,154.421
C01364=1077.961,225.156,-79.921,174.717,25.617,154.421
C01365=1077.955,224.907,-79.895,174.715,25.614,154.420
C01366=1077.950,224.658,-79.869,174.712,25.610,154.420
C01367=1077.944,224.409,-79.843,174.709,25.606,154.419
C01368=1077.938,224.160,-79.818,174.707,25.603,154.419
C01369=1077.933,223.912,-79.793,174.705,25.600,154.418
C01370=1077.927,223.663,-79.767,174.703,25.596,154.418
C01371=1077.921,223.415,-79.741,174.701,25.592,154.417
C01372=1077.916,223.166,-79.715,174.698,25.588,154.417
C01373=1077.906,222.757,-79.673,174.694,25.582,154.416
C01374=1077.897,222.347,-79.630,174.691,25.576,154.415
C01375=1077.887,221.937,-79.588,174.687,25.571,154.414
C01376=1077.879,221.528,-79.546,174.683,25.565,154.414
C01377=1077.872,221.279,-79.521,174.680,25.561,154.413
C01378=1077.867,221.030,-79.496,174.678,25.558,154.413
C01379=1077.861,220.781,-79.470,174.676,25.554,154.412
C01380=1077.855,220.533,-79.445,174.674,25.551,154.412
C01381=1077.849,220.284,-79.420,174.672,25.547,154.411
C01382=1077.844,220.035,-79.394,174.670,25.543,154.411
C01383=1077.838,219.787,-79.369,174.667,25.540,154.410
C01384=1077.832,219.539,-79.344,174.664,25.536,154.410
C01385=1077.827,219.290,-79.318,174.662,25.533,154.409
C01386=1077.820,219.041,-79.293,174.660,25.529,154.409
C01387=1077.814,218.792,-79.267,174.658,25.526,154.408
C01388=1077.810,218.543,-79.242,174.656,25.522,154.408
C01389=1077.803,218.295,-79.217,174.654,25.519,154.407
C01390=1077.797,218.046,-79.192,174.651,25.515,154.407
C01391=1077.792,217.798,-79.166,174.648,25.511,154.406
C01392=1077.786,217.549,-79.141,174.646,25.508,154.406
C01393=1077.780,217.300,-79.116,174.644,25.504,154.405
C01394=1077.775,217.052,-79.091,174.642,25.501,154.405
C01395=1077.769,216.803,-79.065,174.640,25.497,154.404
C01396=1077.763,216.554,-79.040,174.638,25.494,154.404
C01397=1077.757,216.306,-79.015,174.636,25.490,154.403
C01398=1077.752,216.057,-78.990,174.633,25.486,154.403
C01399=1077.746,215.808,-78.964,174.631,25.483,154.402
C01400=1077.740,215.560,-78.939,174.628,25.479,154.402
C01401=1077.734,215.311,-78.915,174.626,25.476,154.401
C01402=1077.729,215.062,-78.889,174.624,25.472,154.401
C01403=1077.723,214.814,-78.864,174.622,25.468,154.400
C01404=1077.717,214.564,-78.839,174.620,25.465,154.400
C01405=1077.712,214.317,-78.814,174.617,25.462,154.399
C01406=1077.706,214.068,-78.788,174.615,25.458,154.399
C01407=1077.700,213.818,-78.764,174.613,25.454,154.398
C01408=1077.695,213.570,-78.739,174.611,25.451,154.398
C01409=1077.689,213.321,-78.714,174.608,25.447,154.397
C01410=1077.684,213.073,-78.689,174.606,25.443,154.397
C01411=1077.678,212.824,-78.663,174.604,25.440,154.396
C01412=1077.672,212.575,-78.639,174.602,25.436,154.396
C01413=1077.666,212.327,-78.614,174.600,25.432,154.395
C01414=1077.661,212.077,-78.589,174.598,25.429,154.395
C01415=1077.655,211.830,-78.564,174.595,25.426,154.394
C01416=1077.649,211.580,-78.539,174.593,25.422,154.394
C01417=1077.643,211.332,-78.514,174.591,25.418,154.393
C01418=1077.637,211.083,-78.490,174.589,25.415,154.393
C01419=1077.632,210.835,-78.465,174.587,25.412,154.392
C01420=1077.626,210.586,-78.440,174.584,25.408,154.392
C01421=1077.620,210.336,-78.416,174.582,25.404,154.391
C01422=1077.615,210.088,-78.390,174.580,25.400,154.391
C01423=1077.609,209.839,-78.365,174.577,25.397,154.390
C01424=1077.604,209.591,-78.340,174.575,25.393,154.390
C01425=1077.594,209.185,-78.300,174.572,25.387,154.389
C01426=1077.585,208.780,-78.260,174.568,25.381,154.388
C01427=1077.576,208.374,-78.220,174.565,25.376,154.388
C01428=1077.566,207.969,-78.179,174.561,25.370,154.387
C01429=1077.542,206.932,-78.080,174.451,25.312,154.388
C01430=1077.537,206.683,-78.056,174.449,25.309,154.387
C01431=1077.531,206.435,-78.031,174.447,25.307,154.387
C01432=1077.526,206.186,-78.007,174.444,25.304,154.387
C01433=1077.520,205.937,-77.983,174.442,25.301,154.386
C01434=1077.514,205.689,-77.959,174.440,25.298,154.386
C01435=1077.509,205.439,-77.935,174.437,25.296,154.386
C01436=1077.503,205.191,-77.912,174.435,25.293,154.386
C01437=1077.497,204.942,-77.887,174.433,25.290,154.385
C01438=1077.492,204.693,-77.863,174.430,25.288,154.385
C01439=1077.486,204.445,-77.839,174.428,25.285,154.385
C01440=1077.481,204.196,-77.815,174.426,25.283,154.384
C01441=1077.476,203.947,-77.791,174.423,25.280,154.384
C01442=1077.469,203.698,-77.767,174.421,25.277,154.384
C01443=1077.464,203.449,-77.744,174.419,25.275,154.384
C01444=1077.459,203.200,-77.719,174.416,25.272,154.383
C01445=1077.453,202.952,-77.696,174.414,25.269,154.383
C01446=1077.447,202.704,-77.671,174.412,25.267,154.383
C01447=1077.442,202.454,-77.648,174.409,25.264,154.383
C01448=1077.436,202.205,-77.624,174.407,25.262,154.382
C01449=1077.430,201.956,-77.601,174.404,25.259,154.382
C01450=1077.425,201.708,-77.577,174.402,25.256,154.382
C01451=1077.418,201.459,-77.553,174.401,25.255,154.382
C01452=1077.413,201.210,-77.529,174.398,25.252,154.381
C01453=1077.407,200.961,-77.505,174.396,25.249,154.381
C01454=1077.402,200.712,-77.482,174.394,25.247,154.381
C01455=1077.396,200.464,-77.458,174.391,25.244,154.381
C01456=1077.389,200.215,-77.434,174.389,25.241,154.380
C01457=1077.384,199.966,-77.411,174.386,25.239,154.380
C01458=1077.378,199.718,-77.387,174.384,25.236,154.380
C01459=1077.373,199.468,-77.363,174.382,25.234,154.379
C01460=1077.367,199.220,-77.340,174.379,25.231,154.379
C01461=1077.362,198.971,-77.317,174.377,25.229,154.379
C01462=1077.356,198.722,-77.292,174.375,25.226,154.379
C01463=1077.350,198.473,-77.269,174.372,25.224,154.379
C01464=1077.344,198.225,-77.246,174.370,25.221,154.378
C01465=1077.339,197.975,-77.222,174.368,25.219,154.378
C01466=1077.333,197.727,-77.198,174.366,25.216,154.378
C01467=1077.328,197.478,-77.175,174.364,25.213,154.377
C01468=1077.322,197.229,-77.152,174.361,25.211,154.377
C01469=1077.316,196.980,-77.128,174.359,25.208,154.377
C01470=1077.311,196.731,-77.104,174.357,25.206,154.377
C01471=1077.305,196.483,-77.081,174.354,25.203,154.376
C01472=1077.299,196.234,-77.058,174.352,25.200,154.376
C01473=1077.294,195.984,-77.034,174.349,25.198,154.376
C01474=1077.288,195.736,-77.011,174.347,25.196,154.376
C01475=1077.282,195.487,-76.988,174.346,25.193,154.375
C01476=1077.277,195.238,-76.964,174.343,25.191,154.375
C01477=1077.271,194.990,-76.940,174.341,25.188,154.375
C01478=1077.265,194.741,-76.917,174.339,25.185,154.375
C01479=1077.260,194.492,-76.894,174.336,25.183,154.374
C01480=1077.254,194.243,-76.870,174.334,25.180,154.374
C01481=1077.249,193.995,-76.847,174.332,25.177,154.374
C01482=1077.244,193.745,-76.824,174.329,25.175,154.374
C01483=1077.237,193.497,-76.800,174.328,25.173,154.373
C01484=1077.232,193.248,-76.777,174.325,25.170,154.373
C01485=1077.226,192.999,-76.754,174.323,25.167,154.373
C01486=1077.221,192.750,-76.731,174.321,25.165,154.372
C01487=1077.215,192.502,-76.707,174.318,25.162,154.372
C01488=1077.209,192.253,-76.684,174.316,25.159,154.372
C01489=1077.204,192.004,-76.661,174.314,25.157,154.372
C01490=1077.198,191.724,-76.634,174.311,25.154,154.371
C01491=1077.192,191.443,-76.608,174.309,25.151,154.371
C01492=1077.185,191.162,-76.582,174.307,25.148,154.371
C01493=1077.179,190.882,-76.556,174.305,25.146,154.370
C01494=1077.173,190.633,-76.533,174.302,25.143,154.370
C01495=1077.168,190.384,-76.510,174.300,25.140,154.370
C01496=1077.162,190.135,-76.487,174.297,25.138,154.370
C01497=1077.157,189.886,-76.463,174.295,25.135,154.369
C01498=1077.151,189.637,-76.440,174.293,25.132,154.369
C01499=1077.145,189.388,-76.417,174.291,25.130,154.369
C01500=1077.140,189.139,-76.394,174.289,25.128,154.369
C01501=1077.134,188.890,-76.371,174.287,25.125,154.368
C01502=1077.129,188.641,-76.348,174.284,25.122,154.368
C01503=1077.123,188.393,-76.324,174.282,25.120,154.368
C01504=1077.117,188.144,-76.301,174.280,25.117,154.368
C01505=1077.112,187.896,-76.279,174.278,25.115,154.367
C01506=1077.107,187.647,-76.255,174.276,25.112,154.367
C01507=1077.101,187.398,-76.232,174.274,25.109,154.367
C01508=1077.096,187.149,-76.209,174.271,25.107,154.366
C01509=1077.090,186.900,-76.186,174.269,25.104,154.366
C01510=1077.084,186.651,-76.163,174.267,25.102,154.366
C01511=1077.079,186.401,-76.141,174.265,25.099,154.366
C01512=1077.074,186.153,-76.118,174.263,25.097,154.365
C01513=1077.069,185.904,-76.095,174.260,25.094,154.365
C01514=1077.063,185.655,-76.072,174.258,25.091,154.365
C01515=1077.057,185.406,-76.049,174.257,25.089,154.365
C01516=1077.052,185.157,-76.026,174.254,25.086,154.364
C01517=1077.046,184.908,-76.003,174.252,25.084,154.364
C01518=1077.041,184.659,-75.980,174.249,25.082,154.364
C01519=1077.034,184.411,-75.957,174.247,25.079,154.364
C01520=1077.029,184.163,-75.935,174.246,25.077,154.363
C01521=1077.024,183.913,-75.913,174.243,25.074,154.363
C01522=1077.018,183.664,-75.890,174.241,25.072,154.363
C01523=1077.012,183.415,-75.867,174.239,25.069,154.363
C01524=1077.006,183.167,-75.844,174.236,25.067,154.362
C01525=1077.000,182.918,-75.821,174.235,25.064,154.362
C01526=1076.995,182.668,-75.799,174.232,25.062,154.362
C01527=1076.989,182.419,-75.776,174.230,25.060,154.362
C01528=1076.982,182.171,-75.754,174.228,25.057,154.361
C01529=1076.977,181.922,-75.731,174.225,25.054,154.361
C01530=1076.971,181.672,-75.709,174.224,25.052,154.361
C01531=1076.965,181.424,-75.686,174.221,25.050,154.361
C01532=1076.960,181.175,-75.663,174.219,25.047,154.360
C01533=1076.954,180.927,-75.641,174.217,25.045,154.360
C01534=1076.948,180.677,-75.619,174.215,25.042,154.360
C01535=1076.943,180.428,-75.596,174.213,25.040,154.360
C01536=1076.937,180.179,-75.573,174.211,25.037,154.359
C01537=1076.931,179.930,-75.551,174.208,25.035,154.359
C01538=1076.925,179.681,-75.528,174.207,25.032,154.359
C01539=1076.920,179.433,-75.505,174.204,25.030,154.359
C01540=1076.915,179.184,-75.483,174.202,25.027,154.358
C01541=1076.908,178.935,-75.461,174.200,25.025,154.358
C01542=1076.902,178.686,-75.438,174.198,25.023,154.358
C01543=1076.897,178.437,-75.416,174.196,25.020,154.358
C01544=1076.890,178.188,-75.393,174.194,25.017,154.357
C01545=1076.886,177.939,-75.371,174.191,25.015,154.357
C01546=1076.880,177.690,-75.349,174.190,25.013,154.357
C01547=1076.874,177.441,-75.326,174.187,25.010,154.357
C01548=1076.868,177.192,-75.304,174.185,25.008,154.356
C01549=1076.862,176.943,-75.281,174.183,25.005,154.356
C01550=1076.857,176.695,-75.259,174.181,25.003,154.356
C01551=1076.851,176.446,-75.237,174.179,25.000,154.356
C01552=1076.846,176.196,-75.215,174.176,24.998,154.356
C01553=1076.840,175.948,-75.192,174.174,24.995,154.355
C01554=1076.834,175.666,-75.167,174.172,24.993,154.355
C01555=1076.828,175.386,-75.142,174.170,24.990,154.355
C01556=1076.821,175.106,-75.117,174.167,24.987,154.354
C01557=1076.814,174.825,-75.092,174.165,24.984,154.354
C01558=1076.809,174.575,-75.069,174.163,24.982,154.354
C01559=1076.803,174.326,-75.046,174.161,24.979,154.354
C01560=1076.798,174.078,-75.025,174.159,24.977,154.353
C01561=1076.792,173.828,-75.003,174.156,24.974,154.353
C01562=1076.786,173.580,-74.980,174.155,24.972,154.353
C01563=1076.781,173.331,-74.959,174.153,24.970,154.353
C01564=1076.775,173.082,-74.936,174.150,24.967,154.352
C01565=1076.770,172.833,-74.914,174.148,24.964,154.352
C01566=1076.763,172.583,-74.892,174.147,24.962,154.352
C01567=1076.758,172.335,-74.869,174.144,24.959,154.351
C01568=1076.752,172.086,-74.848,174.142,24.957,154.351
C01569=1076.747,171.837,-74.825,174.140,24.954,154.351
C01570=1076.742,171.588,-74.803,174.138,24.952,154.351
C01571=1076.735,171.339,-74.781,174.136,24.949,154.350
C01572=1076.731,171.090,-74.759,174.134,24.947,154.350
C01573=1076.725,170.841,-74.736,174.132,24.945,154.350
C01574=1076.719,170.592,-74.715,174.130,24.942,154.350
C01575=1076.714,170.343,-74.693,174.128,24.940,154.349
C01576=1076.708,170.094,-74.671,174.126,24.937,154.349
C01577=1076.702,169.845,-74.648,174.124,24.934,154.349
C01578=1076.697,169.596,-74.627,174.121,24.932,154.349
C01579=1076.691,169.347,-74.605,174.120,24.929,154.348
C01580=1076.686,169.098,-74.583,174.117,24.927,154.348
C01581=1076.680,168.850,-74.561,174.115,24.924,154.348
C01582=1076.674,168.600,-74.538,174.114,24.922,154.348
C01583=1076.669,168.352,-74.517,174.111,24.919,154.347
C01584=1076.663,168.102,-74.495,174.109,24.916,154.347
C01585=1076.659,167.854,-74.473,174.108,24.915,154.347
C01586=1076.652,167.605,-74.451,174.105,24.912,154.347
C01587=1076.647,167.356,-74.429,174.103,24.909,154.346
C01588=1076.641,167.107,-74.407,174.101,24.907,154.346
C01589=1076.636,166.857,-74.385,174.099,24.904,154.346
C01590=1076.630,166.609,-74.364,174.097,24.902,154.345
C01591=1076.625,166.359,-74.341,174.095,24.899,154.345
C01592=1076.620,166.111,-74.320,174.093,24.897,154.345
C01593=1076.614,165.861,-74.298,174.092,24.894,154.345
C01594=1076.609,165.613,-74.276,174.089,24.892,154.344
C01595=1076.602,165.364,-74.254,174.087,24.889,154.344
C01596=1076.598,165.115,-74.232,174.086,24.887,154.344
C01597=1076.591,164.866,-74.210,174.083,24.884,154.344
C01598=1076.587,164.617,-74.188,174.081,24.881,154.343
C01599=1076.580,164.368,-74.167,174.080,24.879,154.343
C01600=1076.576,164.119,-74.145,174.077,24.876,154.343
C01601=1076.569,163.870,-74.123,174.075,24.874,154.342
C01602=1076.565,163.621,-74.101,174.074,24.872,154.342
C01603=1076.558,163.372,-74.080,174.071,24.869,154.342
C01604=1076.554,163.123,-74.058,174.069,24.866,154.342
C01605=1076.548,162.875,-74.037,174.067,24.864,154.341
C01606=1076.543,162.625,-74.014,174.065,24.861,154.341
C01607=1076.537,162.377,-73.993,174.064,24.859,154.341
C01608=1076.532,162.127,-73.971,174.061,24.856,154.341
C01609=1076.526,161.879,-73.950,174.059,24.854,154.340
C01610=1076.521,161.628,-73.928,174.058,24.851,154.340
C01611=1076.515,161.380,-73.907,174.055,24.849,154.340
C01612=1076.509,161.131,-73.885,174.053,24.846,154.339
C01613=1076.504,160.882,-73.863,174.052,24.844,154.339
C01614=1076.498,160.633,-73.842,174.049,24.841,154.339
C01615=1076.493,160.384,-73.820,174.048,24.839,154.339
C01616=1076.487,160.135,-73.799,174.046,24.836,154.338
C01617=1076.482,159.886,-73.777,174.043,24.834,154.338
C01618=1076.475,159.604,-73.754,174.041,24.831,154.338
C01619=1076.468,159.323,-73.729,174.040,24.828,154.338
C01620=1076.462,159.042,-73.705,174.037,24.826,154.337
C01621=1076.456,158.762,-73.681,174.035,24.823,154.337
C01622=1076.450,158.512,-73.659,174.033,24.820,154.337
C01623=1076.445,158.264,-73.638,174.030,24.818,154.337
C01624=1076.439,158.014,-73.617,174.029,24.815,154.336
C01625=1076.433,157.765,-73.595,174.027,24.813,154.336
C01626=1076.427,157.516,-73.574,174.025,24.810,154.336
C01627=1076.422,157.268,-73.552,174.023,24.808,154.335
C01628=1076.416,157.018,-73.532,174.021,24.805,154.335
C01629=1076.411,156.769,-73.510,174.019,24.803,154.335
C01630=1076.405,156.520,-73.488,174.017,24.800,154.335
C01631=1076.400,156.271,-73.467,174.015,24.798,154.334
C01632=1076.394,156.022,-73.446,174.013,24.796,154.334
C01633=1076.388,155.773,-73.425,174.012,24.793,154.334
C01634=1076.382,155.524,-73.403,174.009,24.791,154.334
C01635=1076.376,155.275,-73.382,174.007,24.788,154.333
C01636=1076.371,155.026,-73.361,174.006,24.786,154.333
C01637=1076.366,154.777,-73.340,174.003,24.783,154.333
C01638=1076.360,154.527,-73.318,174.002,24.781,154.332
C01639=1076.355,154.279,-73.297,173.999,24.778,154.332
C01640=1076.349,154.029,-73.276,173.997,24.775,154.332
C01641=1076.343,153.781,-73.255,173.996,24.773,154.332
C01642=1076.338,153.532,-73.234,173.993,24.771,154.332
C01643=1076.332,153.282,-73.213,173.992,24.768,154.331
C01644=1076.326,153.034,-73.191,173.990,24.766,154.331
C01645=1076.320,152.784,-73.170,173.988,24.763,154.331
C01646=1076.315,152.535,-73.149,173.986,24.761,154.330
C01647=1076.310,152.286,-73.129,173.984,24.758,154.330
C01648=1076.303,152.037,-73.107,173.982,24.756,154.330
C01649=1076.298,151.788,-73.086,173.980,24.753,154.330
C01650=1076.293,151.539,-73.065,173.978,24.751,154.329
C01651=1076.287,151.290,-73.044,173.976,24.748,154.329
C01652=1076.281,151.041,-73.023,173.975,24.746,154.329
C01653=1076.276,150.792,-73.002,173.972,24.744,154.329
C01654=1076.270,150.543,-72.981,173.971,24.741,154.328
C01655=1076.265,150.294,-72.960,173.969,24.739,154.328
C01656=1076.259,150.045,-72.939,173.967,24.736,154.328
C01657=1076.253,149.795,-72.918,173.965,24.734,154.328
C01658=1076.248,149.547,-72.897,173.963,24.731,154.327
C01659=1076.242,149.298,-72.877,173.961,24.729,154.327
C01660=1076.235,149.049,-72.855,173.959,24.726,154.327
C01661=1076.230,148.800,-72.835,173.957,24.724,154.326
C01662=1076.225,148.551,-72.814,173.955,24.721,154.326
C01663=1076.219,148.301,-72.792,173.954,24.719,154.326
C01664=1076.213,148.052,-72.772,173.951,24.716,154.326
C01665=1076.208,147.804,-72.751,173.950,24.714,154.325
C01666=1076.203,147.555,-72.730,173.948,24.712,154.325
C01667=1076.196,147.305,-72.710,173.946,24.709,154.325
C01668=1076.190,147.057,-72.688,173.944,24.707,154.325
C01669=1076.185,146.808,-72.668,173.943,24.704,154.324
C01670=1076.179,146.558,-72.647,173.940,24.702,154.324
C01671=1076.174,146.309,-72.626,173.938,24.699,154.324
C01672=1076.168,146.060,-72.606,173.937,24.697,154.324
C01673=1076.162,145.811,-72.585,173.934,24.694,154.323
C01674=1076.157,145.561,-72.564,173.933,24.692,154.323
C01675=1076.151,145.313,-72.543,173.931,24.689,154.323
C01676=1076.145,145.064,-72.523,173.929,24.687,154.323
C01677=1076.139,144.814,-72.502,173.927,24.684,154.322
C01678=1076.134,144.565,-72.482,173.925,24.682,154.322
C01679=1076.128,144.317,-72.460,173.923,24.679,154.322
C01680=1076.122,144.068,-72.440,173.922,24.677,154.321
C01681=1076.117,143.818,-72.419,173.919,24.674,154.321
C01682=1076.111,143.537,-72.396,173.917,24.672,154.321
C01683=1076.104,143.255,-72.373,173.916,24.669,154.321
C01684=1076.098,142.974,-72.350,173.913,24.666,154.320
C01685=1076.092,142.693,-72.327,173.911,24.663,154.320
C01686=1076.085,142.443,-72.305,173.909,24.661,154.320
C01687=1076.080,142.194,-72.284,173.907,24.658,154.319
C01688=1076.074,141.946,-72.264,173.905,24.656,154.319
C01689=1076.069,141.696,-72.244,173.904,24.653,154.319
C01690=1076.064,141.447,-72.223,173.901,24.651,154.319
C01691=1076.058,141.198,-72.203,173.900,24.648,154.318
C01692=1076.052,140.949,-72.183,173.899,24.646,154.318
C01693=1076.047,140.700,-72.162,173.896,24.643,154.318
C01694=1076.041,140.450,-72.141,173.895,24.641,154.318
C01695=1076.035,140.202,-72.121,173.893,24.638,154.317
C01696=1076.030,139.953,-72.100,173.891,24.636,154.317
C01697=1076.023,139.704,-72.080,173.889,24.633,154.317
C01698=1076.018,139.454,-72.059,173.888,24.631,154.316
C01699=1076.013,139.205,-72.039,173.885,24.628,154.316
C01700=1076.007,138.957,-72.019,173.884,24.626,154.316
C01701=1076.001,138.707,-71.998,173.882,24.623,154.316
C01702=1075.995,138.458,-71.978,173.880,24.621,154.315
C01703=1075.990,138.209,-71.957,173.878,24.618,154.315
C01704=1075.984,137.960,-71.937,173.877,24.616,154.315
C01705=1075.978,137.711,-71.917,173.874,24.613,154.315
C01706=1075.973,137.462,-71.896,173.873,24.611,154.314
C01707=1075.967,137.213,-71.876,173.871,24.608,154.314
C01708=1075.961,136.963,-71.855,173.869,24.606,154.314
C01709=1075.955,136.714,-71.835,173.867,24.604,154.314
C01710=1075.950,136.465,-71.815,173.865,24.601,154.313
C01711=1075.944,136.216,-71.795,173.863,24.599,154.313
C01712=1075.939,135.967,-71.775,173.862,24.596,154.313
C01713=1075.933,135.718,-71.755,173.859,24.594,154.312
C01714=1075.928,135.469,-71.735,173.858,24.591,154.312
C01715=1075.922,135.220,-71.715,173.857,24.589,154.312
C01716=1075.916,134.970,-71.694,173.854,24.586,154.312
C01717=1075.910,134.721,-71.674,173.853,24.584,154.311
C01718=1075.905,134.472,-71.653,173.851,24.581,154.311
C01719=1075.899,134.223,-71.633,173.849,24.579,154.311
C01720=1075.893,133.974,-71.614,173.847,24.576,154.310
C01721=1075.888,133.725,-71.593,173.846,24.574,154.310
C01722=1075.882,133.476,-71.573,173.843,24.571,154.310
C01723=1075.876,133.227,-71.553,173.842,24.569,154.310
C01724=1075.870,132.978,-71.533,173.840,24.566,154.309
C01725=1075.865,132.729,-71.512,173.838,24.564,154.309
C01726=1075.860,132.479,-71.493,173.837,24.562,154.309
C01727=1075.854,132.230,-71.473,173.834,24.559,154.309
C01728=1075.848,131.981,-71.452,173.833,24.557,154.308
C01729=1075.842,131.732,-71.432,173.831,24.554,154.308
C01730=1075.837,131.482,-71.412,173.829,24.552,154.308
C01731=1075.831,131.233,-71.393,173.827,24.549,154.307
C01732=1075.825,130.985,-71.373,173.826,24.547,154.307
C01733=1075.819,130.736,-71.353,173.823,24.544,154.307
C01734=1075.814,130.486,-71.333,173.822,24.542,154.307
C01735=1075.808,130.237,-71.313,173.821,24.539,154.306
C01736=1075.802,129.988,-71.293,173.818,24.537,154.306
C01737=1075.796,129.738,-71.273,173.817,24.534,154.306
C01738=1075.790,129.489,-71.253,173.815,24.532,154.306
C01739=1075.784,129.240,-71.233,173.813,24.530,154.305
C01740=1075.779,128.991,-71.213,173.811,24.527,154.305
C01741=1075.773,128.742,-71.194,173.809,24.525,154.305
C01742=1075.767,128.493,-71.174,173.808,24.522,154.305
C01743=1075.761,128.244,-71.154,173.806,24.520,154.304
C01744=1075.756,127.995,-71.134,173.804,24.517,154.304
C01745=1075.750,127.745,-71.115,173.802,24.515,154.304
C01746=1075.743,127.465,-71.092,173.801,24.512,154.303
C01747=1075.737,127.182,-71.069,173.799,24.509,154.303
C01748=1075.730,126.902,-71.047,173.796,24.506,154.303
C01749=1075.723,126.620,-71.025,173.794,24.503,154.302
C01750=1075.718,126.370,-71.005,173.793,24.501,154.302
C01751=1075.712,126.121,-70.985,173.791,24.499,154.302
C01752=1075.706,125.872,-70.965,173.789,24.496,154.302
C01753=1075.701,125.623,-70.946,173.788,24.494,154.301
C01754=1075.695,125.374,-70.926,173.785,24.491,154.301
C01755=1075.689,125.125,-70.907,173.784,24.489,154.301
C01756=1075.684,124.875,-70.886,173.783,24.487,154.301
C01757=1075.678,124.626,-70.867,173.780,24.483,154.300
C01758=1075.672,124.377,-70.847,173.779,24.481,154.300
C01759=1075.666,124.128,-70.828,173.777,24.478,154.300
C01760=1075.660,123.879,-70.808,173.775,24.476,154.299
C01761=1075.655,123.630,-70.789,173.773,24.473,154.299
C01762=1075.650,123.380,-70.769,173.772,24.471,154.299
C01763=1075.644,123.131,-70.749,173.770,24.469,154.298
C01764=1075.638,122.882,-70.729,173.768,24.466,154.298
C01765=1075.633,122.633,-70.710,173.767,24.463,154.298
C01766=1075.627,122.384,-70.691,173.765,24.461,154.298
C01767=1075.621,122.135,-70.671,173.763,24.458,154.297
C01768=1075.615,121.886,-70.651,173.762,24.456,154.297
C01769=1075.610,121.636,-70.632,173.759,24.453,154.297
C01770=1075.604,121.387,-70.612,173.758,24.451,154.297
C01771=1075.599,121.138,-70.592,173.757,24.449,154.296
C01772=1075.593,120.888,-70.573,173.754,24.446,154.296
C01773=1075.587,120.640,-70.553,173.753,24.444,154.296
C01774=1075.581,120.390,-70.534,173.751,24.441,154.295
C01775=1075.575,120.141,-70.514,173.749,24.439,154.295
C01776=1075.570,119.893,-70.495,173.748,24.436,154.295
C01777=1075.565,119.643,-70.476,173.746,24.433,154.295
C01778=1075.559,119.394,-70.457,173.744,24.431,154.294
C01779=1075.553,119.145,-70.437,173.742,24.428,154.294
C01780=1075.548,118.895,-70.417,173.741,24.426,154.294
C01781=1075.542,118.646,-70.398,173.739,24.423,154.293
C01782=1075.536,118.397,-70.378,173.737,24.421,154.293
C01783=1075.531,118.148,-70.359,173.736,24.418,154.293
C01784=1075.525,117.899,-70.340,173.734,24.416,154.293
C01785=1075.520,117.649,-70.320,173.732,24.413,154.292
C01786=1075.514,117.400,-70.300,173.731,24.410,154.292
C01787=1075.508,117.151,-70.281,173.729,24.408,154.292
C01788=1075.502,116.902,-70.262,173.727,24.405,154.291
C01789=1075.497,116.653,-70.243,173.726,24.403,154.291
C01790=1075.492,116.403,-70.224,173.724,24.400,154.291
C01791=1075.486,116.155,-70.204,173.722,24.398,154.290
C01792=1075.480,115.905,-70.185,173.721,24.395,154.290
C01793=1075.474,115.656,-70.165,173.719,24.392,154.290
C01794=1075.469,115.407,-70.146,173.717,24.390,154.290
C01795=1075.463,115.158,-70.127,173.716,24.388,154.289
C01796=1075.457,114.909,-70.107,173.714,24.385,154.289
C01797=1075.452,114.659,-70.088,173.712,24.383,154.289
C01798=1075.447,114.410,-70.068,173.711,24.380,154.288
C01799=1075.441,114.161,-70.050,173.709,24.377,154.288
